LIN {X 0,Y 293.963,Z 864.101,A -85,B 0,C 180,E1 22484.69,E2 22484.69} C_VEL
LIN {X 0,Y 291.731,Z 885.512,A -85,B 0,C 180,E1 22491.042,E2 22491.042} C_VEL
LIN {X 0,Y 291.359,Z 899.593,A -85,B 0,C 180,E1 22497.023,E2 22497.023} C_VEL
LIN {X 0,Y 292.208,Z 908.654,A -85,B 0,C 180,E1 22502.975,E2 22502.975} C_VEL
LIN {X 0,Y 295.422,Z 913.131,A -85,B 0,C 180,E1 22508.853,E2 22508.853} C_VEL
LIN {X 0,Y 300.698,Z 913.398,A -85,B 0,C 180,E1 22514.593,E2 22514.593} C_VEL
LIN {X 0,Y 310.967,Z 908.328,A -85,B 0,C 180,E1 22521.434,E2 22521.434} C_VEL
LIN {X 0,Y 325.668,Z 897.626,A -85,B 0,C 180,E1 22527.724,E2 22527.724} C_VEL
LIN {X 0,Y 349.66,Z 878.572,A -85,B 0,C 180,E1 22534.282,E2 22534.282} C_VEL
LIN {X 0,Y 365.291,Z 866.098,A -85,B 0,C 180,E1 22537.259,E2 22537.259} C_VEL
LIN {X 0,Y 331.443,Z 903.67,A -85,B 0,C 180,E1 22545.054,E2 22545.054} C_VEL
LIN {X 0,Y 310.197,Z 930.316,A -85,B 0,C 180,E1 22553.256,E2 22553.256} C_VEL
LIN {X 0,Y 296.493,Z 951.276,A -85,B 0,C 180,E1 22562.626,E2 22562.626} C_VEL
LIN {X 0,Y 290.643,Z 964.921,A -85,B 0,C 180,E1 22571.781,E2 22571.781} C_VEL
LIN {X 0,Y 289.464,Z 970.796,A -85,B 0,C 180,E1 22577.922,E2 22577.922} C_VEL
LIN {X 0,Y 289.713,Z 973.891,A -85,B 0,C 180,E1 22584.004,E2 22584.004} C_VEL
LIN {X 0,Y 290.557,Z 973.915,A -85,B 0,C 180,E1 22590.008,E2 22590.008} C_VEL
LIN {X 0,Y 290.157,Z 969.252,A -85,B 0,C 180,E1 22597.235,E2 22597.235} C_VEL
LIN {X 0,Y 290.402,Z 960.92,A -85,B 0,C 180,E1 22605.131,E2 22605.131} C_VEL
LIN {X 0,Y 292.996,Z 947.16,A -85,B 0,C 180,E1 22612.83,E2 22612.83} C_VEL
LIN {X 0,Y 298.847,Z 927.81,A -85,B 0,C 180,E1 22620.054,E2 22620.054} C_VEL
LIN {X 0,Y 307.221,Z 903.866,A -85,B 0,C 180,E1 22626.297,E2 22626.297} C_VEL
LIN {X 0,Y 316.929,Z 875.444,A -85,B 0,C 180,E1 22631.566,E2 22631.566} C_VEL
LIN {X 0,Y 326.727,Z 843.194,A -85,B 0,C 180,E1 22635.791,E2 22635.791} C_VEL
LIN {X 0,Y 335.469,Z 807.511,A -85,B 0,C 180,E1 22639.019,E2 22639.019} C_VEL
LIN {X 0,Y 345.478,Z 755.854,A -85,B 0,C 180,E1 22642.286,E2 22642.286} C_VEL
LIN {X 0,Y 347.447,Z 742.622,A -85,B 0,C 180,E1 22643.014,E2 22643.014} C_VEL
LIN {X 0,Y 330.365,Z 668.326,A -85,B 0,C 180,E1 22652.795,E2 22652.795} C_VEL
LIN {X 0,Y 328.166,Z 660.053,A -85,B 0,C 180,E1 22654.078,E2 22654.078} C_VEL
LIN {X 0,Y 318.814,Z 645.104,A -85,B 0,C 180,E1 22658.71,E2 22658.71} C_VEL
LIN {X 0,Y 315.788,Z 643.613,A -85,B 0,C 180,E1 22660.163,E2 22660.163} C_VEL
LIN {X 0,Y 310.485,Z 643.76,A -85,B 0,C 180,E1 22662.744,E2 22662.744} C_VEL
LIN {X 0,Y 306.565,Z 637.974,A -85,B 0,C 180,E1 22665.692,E2 22665.692} C_VEL
LIN {X 0,Y 302.237,Z 631.324,A -85,B 0,C 180,E1 22669.893,E2 22669.893} C_VEL
LIN {X 0,Y 298.732,Z 625.168,A -85,B 0,C 180,E1 22675.361,E2 22675.361} C_VEL
LIN {X 0,Y 297.1,Z 623.883,A -85,B 0,C 180,E1 22683.651,E2 22683.651} C_VEL
LIN {X 0,Y 298.132,Z 625.461,A -85,B 0,C 180,E1 22687.753,E2 22687.753} C_VEL
LIN {X 0,Y 301.609,Z 631.309,A -85,B 0,C 180,E1 22693.761,E2 22693.761} C_VEL
LIN {X 0,Y 306.971,Z 640.946,A -85,B 0,C 180,E1 22699.364,E2 22699.364} C_VEL
LIN {X 0,Y 313.809,Z 652.315,A -85,B 0,C 180,E1 22704.391,E2 22704.391} C_VEL
LIN {X 0,Y 324.604,Z 672.136,A -85,B 0,C 180,E1 22710.592,E2 22710.592} C_VEL
LIN {X 0,Y 335.868,Z 696.454,A -85,B 0,C 180,E1 22715.988,E2 22715.988} C_VEL
LIN {X 0,Y 344.416,Z 721.512,A -85,B 0,C 180,E1 22720.282,E2 22720.282} C_VEL
LIN {X 0,Y 347.289,Z 737.002,A -85,B 0,C 180,E1 22722.591,E2 22722.591} C_VEL
LIN {X 0,Y 337.653,Z 771.94,A -85,B 0,C 180,E1 22725.601,E2 22725.601} C_VEL
LIN {X 0,Y 326.46,Z 803.597,A -85,B 0,C 180,E1 22729.465,E2 22729.465} C_VEL
LIN {X 0,Y 314.714,Z 831.598,A -85,B 0,C 180,E1 22734.275,E2 22734.275} C_VEL
LIN {X 0,Y 303.549,Z 855.386,A -85,B 0,C 180,E1 22740.046,E2 22740.046} C_VEL
LIN {X 0,Y 294.509,Z 873.806,A -85,B 0,C 180,E1 22746.493,E2 22746.493} C_VEL
LIN {X 0,Y 287.852,Z 887.888,A -85,B 0,C 180,E1 22753.949,E2 22753.949} C_VEL
LIN {X 0,Y 284.529,Z 895.556,A -85,B 0,C 180,E1 22760.799,E2 22760.799} C_VEL
LIN {X 0,Y 283.36,Z 898.747,A -85,B 0,C 180,E1 22766.926,E2 22766.926} C_VEL
LIN {X 0,Y 283.471,Z 898.702,A -85,B 0,C 180,E1 22773.056,E2 22773.056} C_VEL
LIN {X 0,Y 285.219,Z 893.795,A -85,B 0,C 180,E1 22781.036,E2 22781.036} C_VEL
LIN {X 0,Y 290.075,Z 882.965,A -85,B 0,C 180,E1 22788.94,E2 22788.94} C_VEL
LIN {X 0,Y 297.256,Z 868.058,A -85,B 0,C 180,E1 22795.666,E2 22795.666} C_VEL
LIN {X 0,Y 307.265,Z 847.474,A -85,B 0,C 180,E1 22802.004,E2 22802.004} C_VEL
LIN {X 0,Y 319.289,Z 820.866,A -85,B 0,C 180,E1 22807.652,E2 22807.652} C_VEL
LIN {X 0,Y 331.221,Z 790.376,A -85,B 0,C 180,E1 22812.204,E2 22812.204} C_VEL
LIN {X 0,Y 342.367,Z 755.645,A -85,B 0,C 180,E1 22815.832,E2 22815.832} C_VEL
LIN {X 0,Y 347.152,Z 734.437,A -85,B 0,C 180,E1 22817.597,E2 22817.597} C_VEL
LIN {X 0,Y 340.844,Z 709.744,A -85,B 0,C 180,E1 22821.525,E2 22821.525} C_VEL
LIN {X 0,Y 338.651,Z 705.006,A -85,B 0,C 180,E1 22822.452,E2 22822.452} C_VEL
LIN {X 0,Y 327.156,Z 719.096,A -85,B 0,C 180,E1 22823.933,E2 22823.933} C_VEL
LIN {X 0,Y 319.775,Z 728.865,A -85,B 0,C 180,E1 22824.78,E2 22824.78} C_VEL
LIN {X 0,Y 316.357,Z 731.37,A -85,B 0,C 180,E1 22825.427,E2 22825.427} C_VEL
LIN {X 0,Y 310.131,Z 739.58,A -85,B 0,C 180,E1 22826.143,E2 22826.143} C_VEL
LIN {X 0,Y 305.98,Z 742.075,A -85,B 0,C 180,E1 22827.121,E2 22827.121} C_VEL
LIN {X 0,Y 299.689,Z 781.3,A -85,B 0,C 180,E1 22830.684,E2 22830.684} C_VEL
LIN {X 0,Y 293.509,Z 817.551,A -85,B 0,C 180,E1 22835.353,E2 22835.353} C_VEL
LIN {X 0,Y 288.411,Z 848.674,A -85,B 0,C 180,E1 22840.89,E2 22840.89} C_VEL
LIN {X 0,Y 284.991,Z 873.356,A -85,B 0,C 180,E1 22846.948,E2 22846.948} C_VEL
LIN {X 0,Y 283.545,Z 891.452,A -85,B 0,C 180,E1 22853.1,E2 22853.1} C_VEL
LIN {X 0,Y 283.712,Z 905.176,A -85,B 0,C 180,E1 22860.004,E2 22860.004} C_VEL
LIN {X 0,Y 285.808,Z 912.321,A -85,B 0,C 180,E1 22866.089,E2 22866.089} C_VEL
LIN {X 0,Y 290.137,Z 915.158,A -85,B 0,C 180,E1 22872.059,E2 22872.059} C_VEL
LIN {X 0,Y 296.986,Z 913.91,A -85,B 0,C 180,E1 22877.825,E2 22877.825} C_VEL
LIN {X 0,Y 309.514,Z 907.303,A -85,B 0,C 180,E1 22884.588,E2 22884.588} C_VEL
LIN {X 0,Y 328.712,Z 894.071,A -85,B 0,C 180,E1 22891.233,E2 22891.233} C_VEL
LIN {X 0,Y 355.231,Z 874.877,A -85,B 0,C 180,E1 22897.074,E2 22897.074} C_VEL
LIN {X 0,Y 355.139,Z 875.264,A -85,B 0,C 180,E1 22897.5,E2 22897.5} C_VEL
LIN {X 0,Y 325.035,Z 906.212,A -85,B 0,C 180,E1 22904.36,E2 22904.36} C_VEL
LIN {X 0,Y 302.368,Z 932.529,A -85,B 0,C 180,E1 22913.044,E2 22913.044} C_VEL
LIN {X 0,Y 288.301,Z 952.616,A -85,B 0,C 180,E1 22922.819,E2 22922.819} C_VEL
LIN {X 0,Y 282.424,Z 965.885,A -85,B 0,C 180,E1 22932.847,E2 22932.847} C_VEL
LIN {X 0,Y 281.639,Z 971.637,A -85,B 0,C 180,E1 22940.721,E2 22940.721} C_VEL
LIN {X 0,Y 282.269,Z 973.069,A -85,B 0,C 180,E1 22946.931,E2 22946.931} C_VEL
LIN {X 0,Y 282.753,Z 972.61,A -85,B 0,C 180,E1 22950.008,E2 22950.008} C_VEL
LIN {X 0,Y 282.308,Z 968.072,A -85,B 0,C 180,E1 22957.437,E2 22957.437} C_VEL
LIN {X 0,Y 282.57,Z 959.86,A -85,B 0,C 180,E1 22965.561,E2 22965.561} C_VEL
LIN {X 0,Y 285.43,Z 946.05,A -85,B 0,C 180,E1 22973.471,E2 22973.471} C_VEL
LIN {X 0,Y 291.695,Z 926.652,A -85,B 0,C 180,E1 22980.87,E2 22980.87} C_VEL
LIN {X 0,Y 300.52,Z 902.658,A -85,B 0,C 180,E1 22987.241,E2 22987.241} C_VEL
LIN {X 0,Y 310.747,Z 874.204,A -85,B 0,C 180,E1 22992.585,E2 22992.585} C_VEL
LIN {X 0,Y 320.997,Z 841.931,A -85,B 0,C 180,E1 22996.853,E2 22996.853} C_VEL
LIN {X 0,Y 330.033,Z 806.731,A -85,B 0,C 180,E1 23000.051,E2 23000.051} C_VEL
LIN {X 0,Y 340.278,Z 755.895,A -85,B 0,C 180,E1 23003.286,E2 23003.286} C_VEL
LIN {X 0,Y 341.629,Z 744.601,A -85,B 0,C 180,E1 23003.994,E2 23003.994} C_VEL
LIN {X 0,Y 326.511,Z 673.546,A -85,B 0,C 180,E1 23013.593,E2 23013.593} C_VEL
LIN {X 0,Y 324.558,Z 665.67,A -85,B 0,C 180,E1 23014.887,E2 23014.887} C_VEL
LIN {X 0,Y 314.172,Z 649.402,A -85,B 0,C 180,E1 23020.362,E2 23020.362} C_VEL
LIN {X 0,Y 310.485,Z 643.76,A -85,B 0,C 180,E1 23022.744,E2 23022.744} C_VEL
LIN {X 0,Y 305.445,Z 642.335,A -85,B 0,C 180,E1 23025.87,E2 23025.87} C_VEL
LIN {X 0,Y 301.668,Z 640.672,A -85,B 0,C 180,E1 23028.861,E2 23028.861} C_VEL
LIN {X 0,Y 301.51,Z 640.292,A -85,B 0,C 180,E1 23029.053,E2 23029.053} C_VEL
LIN {X 0,Y 297.03,Z 632.389,A -85,B 0,C 180,E1 23035.884,E2 23035.884} C_VEL
LIN {X 0,Y 296.025,Z 631.913,A -85,B 0,C 180,E1 23045.871,E2 23045.871} C_VEL
LIN {X 0,Y 296.469,Z 633.916,A -85,B 0,C 180,E1 23047.982,E2 23047.982} C_VEL
LIN {X 0,Y 300.315,Z 640.431,A -85,B 0,C 180,E1 23054.409,E2 23054.409} C_VEL
LIN {X 0,Y 304.755,Z 648.592,A -85,B 0,C 180,E1 23059.15,E2 23059.15} C_VEL
LIN {X 0,Y 311.109,Z 659.692,A -85,B 0,C 180,E1 23064.063,E2 23064.063} C_VEL
LIN {X 0,Y 321.105,Z 678.543,A -85,B 0,C 180,E1 23070.055,E2 23070.055} C_VEL
LIN {X 0,Y 331.913,Z 702.757,A -85,B 0,C 180,E1 23075.512,E2 23075.512} C_VEL
LIN {X 0,Y 339.614,Z 727.51,A -85,B 0,C 180,E1 23079.862,E2 23079.862} C_VEL
LIN {X 0,Y 341.411,Z 740.531,A -85,B 0,C 180,E1 23081.817,E2 23081.817} C_VEL
LIN {X 0,Y 331.408,Z 775.162,A -85,B 0,C 180,E1 23084.883,E2 23084.883} C_VEL
LIN {X 0,Y 319.916,Z 806.201,A -85,B 0,C 180,E1 23088.789,E2 23088.789} C_VEL
LIN {X 0,Y 307.632,Z 834.289,A -85,B 0,C 180,E1 23093.759,E2 23093.759} C_VEL
LIN {X 0,Y 295.696,Z 858.447,A -85,B 0,C 180,E1 23099.906,E2 23099.906} C_VEL
LIN {X 0,Y 286.434,Z 876.562,A -85,B 0,C 180,E1 23106.616,E2 23106.616} C_VEL
LIN {X 0,Y 279.777,Z 889.923,A -85,B 0,C 180,E1 23114.28,E2 23114.28} C_VEL
LIN {X 0,Y 276.772,Z 896.554,A -85,B 0,C 180,E1 23120.538,E2 23120.538} C_VEL
LIN {X 0,Y 275.54,Z 899.735,A -85,B 0,C 180,E1 23126.839,E2 23126.839} C_VEL
LIN {X 0,Y 275.65,Z 899.69,A -85,B 0,C 180,E1 23133.142,E2 23133.142} C_VEL
LIN {X 0,Y 277.381,Z 895.05,A -85,B 0,C 180,E1 23141.06,E2 23141.06} C_VEL
LIN {X 0,Y 282.091,Z 885.159,A -85,B 0,C 180,E1 23148.792,E2 23148.792} C_VEL
LIN {X 0,Y 290.171,Z 869.098,A -85,B 0,C 180,E1 23156.341,E2 23156.341} C_VEL
LIN {X 0,Y 301.279,Z 847.128,A -85,B 0,C 180,E1 23163.147,E2 23163.147} C_VEL
LIN {X 0,Y 313.878,Z 820.133,A -85,B 0,C 180,E1 23168.86,E2 23168.86} C_VEL
LIN {X 0,Y 326.366,Z 788.955,A -85,B 0,C 180,E1 23173.438,E2 23173.438} C_VEL
LIN {X 0,Y 337.493,Z 754.65,A -85,B 0,C 180,E1 23176.963,E2 23176.963} C_VEL
LIN {X 0,Y 341.605,Z 738.117,A -85,B 0,C 180,E1 23178.307,E2 23178.307} C_VEL
LIN {X 0,Y 336.717,Z 716.824,A -85,B 0,C 180,E1 23181.789,E2 23181.789} C_VEL
LIN {X 0,Y 335.916,Z 715.7,A -85,B 0,C 180,E1 23182.092,E2 23182.092} C_VEL
LIN {X 0,Y 329.302,Z 723.742,A -85,B 0,C 180,E1 23182.863,E2 23182.863} C_VEL
LIN {X 0,Y 320.621,Z 734.521,A -85,B 0,C 180,E1 23183.806,E2 23183.806} C_VEL
LIN {X 0,Y 314.182,Z 741.259,A -85,B 0,C 180,E1 23184.652,E2 23184.652} C_VEL
LIN {X 0,Y 307.063,Z 747.905,A -85,B 0,C 180,E1 23185.758,E2 23185.758} C_VEL
LIN {X 0,Y 299.477,Z 755.381,A -85,B 0,C 180,E1 23186.895,E2 23186.895} C_VEL
LIN {X 0,Y 296.238,Z 757.549,A -85,B 0,C 180,E1 23187.839,E2 23187.839} C_VEL
LIN {X 0,Y 289.52,Z 796.999,A -85,B 0,C 180,E1 23192.06,E2 23192.06} C_VEL
LIN {X 0,Y 283.552,Z 831.369,A -85,B 0,C 180,E1 23197.216,E2 23197.216} C_VEL
LIN {X 0,Y 278.964,Z 859.516,A -85,B 0,C 180,E1 23203.033,E2 23203.033} C_VEL
LIN {X 0,Y 276.333,Z 881.753,A -85,B 0,C 180,E1 23209.342,E2 23209.342} C_VEL
LIN {X 0,Y 275.548,Z 898.545,A -85,B 0,C 180,E1 23216.063,E2 23216.063} C_VEL
LIN {X 0,Y 276.484,Z 909.926,A -85,B 0,C 180,E1 23223.145,E2 23223.145} C_VEL
LIN {X 0,Y 279.977,Z 915.293,A -85,B 0,C 180,E1 23229.346,E2 23229.346} C_VEL
LIN {X 0,Y 285.775,Z 916.584,A -85,B 0,C 180,E1 23235.374,E2 23235.374} C_VEL
LIN {X 0,Y 296.93,Z 912.826,A -85,B 0,C 180,E1 23242.501,E2 23242.501} C_VEL
LIN {X 0,Y 314.72,Z 902.755,A -85,B 0,C 180,E1 23249.567,E2 23249.567} C_VEL
LIN {X 0,Y 340.531,Z 885.96,A -85,B 0,C 180,E1 23256.034,E2 23256.034} C_VEL
LIN {X 0,Y 346.696,Z 881.931,A -85,B 0,C 180,E1 23257.183,E2 23257.183} C_VEL
LIN {X 0,Y 312.804,Z 914.491,A -85,B 0,C 180,E1 23265.393,E2 23265.393} C_VEL
LIN {X 0,Y 290.43,Z 939.321,A -85,B 0,C 180,E1 23274.989,E2 23274.989} C_VEL
LIN {X 0,Y 278.434,Z 956.654,A -85,B 0,C 180,E1 23285.065,E2 23285.065} C_VEL
LIN {X 0,Y 274.025,Z 967.466,A -85,B 0,C 180,E1 23295.168,E2 23295.168} C_VEL
LIN {X 0,Y 274.019,Z 971.558,A -85,B 0,C 180,E1 23303.659,E2 23303.659} C_VEL
LIN {X 0,Y 274.983,Z 971.26,A -85,B 0,C 180,E1 23310.009,E2 23310.009} C_VEL
LIN {X 0,Y 274.418,Z 966.967,A -85,B 0,C 180,E1 23317.783,E2 23317.783} C_VEL
LIN {X 0,Y 274.735,Z 958.801,A -85,B 0,C 180,E1 23326.016,E2 23326.016} C_VEL
LIN {X 0,Y 277.873,Z 944.933,A -85,B 0,C 180,E1 23334.149,E2 23334.149} C_VEL
LIN {X 0,Y 284.342,Z 926.124,A -85,B 0,C 180,E1 23341.516,E2 23341.516} C_VEL
LIN {X 0,Y 293.926,Z 901.439,A -85,B 0,C 180,E1 23348.225,E2 23348.225} C_VEL
LIN {X 0,Y 304.675,Z 872.948,A -85,B 0,C 180,E1 23353.643,E2 23353.643} C_VEL
LIN {X 0,Y 315.422,Z 840.584,A -85,B 0,C 180,E1 23357.956,E2 23357.956} C_VEL
LIN {X 0,Y 324.619,Z 806.394,A -85,B 0,C 180,E1 23361.084,E2 23361.084} C_VEL
LIN {X 0,Y 335.497,Z 754.329,A -85,B 0,C 180,E1 23364.396,E2 23364.396} C_VEL
LIN {X 0,Y 336.175,Z 747.644,A -85,B 0,C 180,E1 23364.852,E2 23364.852} C_VEL
LIN {X 0,Y 322.845,Z 679.483,A -85,B 0,C 180,E1 23374.297,E2 23374.297} C_VEL
LIN {X 0,Y 320.939,Z 671.429,A -85,B 0,C 180,E1 23375.641,E2 23375.641} C_VEL
LIN {X 0,Y 309.444,Z 652.358,A -85,B 0,C 180,E1 23382.382,E2 23382.382} C_VEL
LIN {X 0,Y 303.923,Z 644.729,A -85,B 0,C 180,E1 23386.576,E2 23386.576} C_VEL
LIN {X 0,Y 301.51,Z 640.292,A -85,B 0,C 180,E1 23389.053,E2 23389.053} C_VEL
LIN {X 0,Y 299.597,Z 640.524,A -85,B 0,C 180,E1 23390.668,E2 23390.668} C_VEL
LIN {X 0,Y 296.515,Z 643.952,A -85,B 0,C 180,E1 23393.147,E2 23393.147} C_VEL
LIN {X 0,Y 296.313,Z 643.797,A -85,B 0,C 180,E1 23393.435,E2 23393.435} C_VEL
LIN {X 0,Y 294.879,Z 639.708,A -85,B 0,C 180,E1 23397.052,E2 23397.052} C_VEL
LIN {X 0,Y 294.554,Z 640.25,A -85,B 0,C 180,E1 23406.919,E2 23406.919} C_VEL
LIN {X 0,Y 298.182,Z 648.151,A -85,B 0,C 180,E1 23414.218,E2 23414.218} C_VEL
LIN {X 0,Y 302.552,Z 656.224,A -85,B 0,C 180,E1 23418.965,E2 23418.965} C_VEL
LIN {X 0,Y 310.3,Z 670.155,A -85,B 0,C 180,E1 23424.995,E2 23424.995} C_VEL
LIN {X 0,Y 320.367,Z 691.113,A -85,B 0,C 180,E1 23431.099,E2 23431.099} C_VEL
LIN {X 0,Y 329.994,Z 715.209,A -85,B 0,C 180,E1 23436.227,E2 23436.227} C_VEL
LIN {X 0,Y 335.936,Z 740.581,A -85,B 0,C 180,E1 23440.621,E2 23440.621} C_VEL
LIN {X 0,Y 332.723,Z 754.359,A -85,B 0,C 180,E1 23441.83,E2 23441.83} C_VEL
LIN {X 0,Y 321.104,Z 789.415,A -85,B 0,C 180,E1 23445.409,E2 23445.409} C_VEL
LIN {X 0,Y 308.323,Z 820.439,A -85,B 0,C 180,E1 23449.981,E2 23449.981} C_VEL
LIN {X 0,Y 295.394,Z 847.143,A -85,B 0,C 180,E1 23455.641,E2 23455.641} C_VEL
LIN {X 0,Y 284.158,Z 868.467,A -85,B 0,C 180,E1 23462.178,E2 23462.178} C_VEL
LIN {X 0,Y 275.343,Z 884.758,A -85,B 0,C 180,E1 23469.727,E2 23469.727} C_VEL
LIN {X 0,Y 270.333,Z 894.669,A -85,B 0,C 180,E1 23477.035,E2 23477.035} C_VEL
LIN {X 0,Y 268.15,Z 899.522,A -85,B 0,C 180,E1 23483.502,E2 23483.502} C_VEL
LIN {X 0,Y 267.775,Z 901.131,A -85,B 0,C 180,E1 23489.991,E2 23489.991} C_VEL
LIN {X 0,Y 268.224,Z 899.464,A -85,B 0,C 180,E1 23496.478,E2 23496.478} C_VEL
LIN {X 0,Y 271.288,Z 892.82,A -85,B 0,C 180,E1 23504.547,E2 23504.547} C_VEL
LIN {X 0,Y 277.595,Z 880.506,A -85,B 0,C 180,E1 23512.453,E2 23512.453} C_VEL
LIN {X 0,Y 287.56,Z 861.943,A -85,B 0,C 180,E1 23519.977,E2 23519.977} C_VEL
LIN {X 0,Y 299.842,Z 838.082,A -85,B 0,C 180,E1 23526.397,E2 23526.397} C_VEL
LIN {X 0,Y 312.256,Z 811.181,A -85,B 0,C 180,E1 23531.438,E2 23531.438} C_VEL
LIN {X 0,Y 324.825,Z 778.911,A -85,B 0,C 180,E1 23535.688,E2 23535.688} C_VEL
LIN {X 0,Y 335.426,Z 743.926,A -85,B 0,C 180,E1 23538.895,E2 23538.895} C_VEL
LIN {X 0,Y 335.302,Z 736.78,A -85,B 0,C 180,E1 23539.849,E2 23539.849} C_VEL
LIN {X 0,Y 332.931,Z 726.038,A -85,B 0,C 180,E1 23541.693,E2 23541.693} C_VEL
LIN {X 0,Y 322.621,Z 738.908,A -85,B 0,C 180,E1 23542.667,E2 23542.667} C_VEL
LIN {X 0,Y 307.588,Z 753.393,A -85,B 0,C 180,E1 23544.646,E2 23544.646} C_VEL
LIN {X 0,Y 298.305,Z 761.782,A -85,B 0,C 180,E1 23546.044,E2 23546.044} C_VEL
LIN {X 0,Y 294.774,Z 764.171,A -85,B 0,C 180,E1 23546.75,E2 23546.75} C_VEL
LIN {X 0,Y 289.618,Z 768.793,A -85,B 0,C 180,E1 23547.569,E2 23547.569} C_VEL
LIN {X 0,Y 286.619,Z 770.796,A -85,B 0,C 180,E1 23548.543,E2 23548.543} C_VEL
LIN {X 0,Y 279.985,Z 808.372,A -85,B 0,C 180,E1 23553.116,E2 23553.116} C_VEL
LIN {X 0,Y 274.281,Z 840.385,A -85,B 0,C 180,E1 23558.541,E2 23558.541} C_VEL
LIN {X 0,Y 270.036,Z 868.042,A -85,B 0,C 180,E1 23564.966,E2 23564.966} C_VEL
LIN {X 0,Y 267.905,Z 889.543,A -85,B 0,C 180,E1 23571.973,E2 23571.973} C_VEL
LIN {X 0,Y 267.866,Z 904.645,A -85,B 0,C 180,E1 23579.194,E2 23579.194} C_VEL
LIN {X 0,Y 270.192,Z 913.939,A -85,B 0,C 180,E1 23586.442,E2 23586.442} C_VEL
LIN {X 0,Y 274.927,Z 917.659,A -85,B 0,C 180,E1 23592.737,E2 23592.737} C_VEL
LIN {X 0,Y 282.404,Z 917.539,A -85,B 0,C 180,E1 23598.779,E2 23598.779} C_VEL
LIN {X 0,Y 295.992,Z 912.372,A -85,B 0,C 180,E1 23605.791,E2 23605.791} C_VEL
LIN {X 0,Y 316.583,Z 901.259,A -85,B 0,C 180,E1 23612.574,E2 23612.574} C_VEL
LIN {X 0,Y 335.318,Z 890.227,A -85,B 0,C 180,E1 23616.783,E2 23616.783} C_VEL
LIN {X 0,Y 336.215,Z 889.95,A -85,B 0,C 180,E1 23617.359,E2 23617.359} C_VEL
LIN {X 0,Y 303.371,Z 919.431,A -85,B 0,C 180,E1 23625.645,E2 23625.645} C_VEL
LIN {X 0,Y 280.056,Z 943.79,A -85,B 0,C 180,E1 23636.33,E2 23636.33} C_VEL
LIN {X 0,Y 269.246,Z 959.185,A -85,B 0,C 180,E1 23646.81,E2 23646.81} C_VEL
LIN {X 0,Y 265.962,Z 967.867,A -85,B 0,C 180,E1 23656.837,E2 23656.837} C_VEL
LIN {X 0,Y 266.156,Z 970.372,A -85,B 0,C 180,E1 23663.471,E2 23663.471} C_VEL
LIN {X 0,Y 267.189,Z 969.885,A -85,B 0,C 180,E1 23670.009,E2 23670.009} C_VEL
LIN {X 0,Y 266.513,Z 965.846,A -85,B 0,C 180,E1 23678.18,E2 23678.18} C_VEL
LIN {X 0,Y 266.947,Z 957.741,A -85,B 0,C 180,E1 23686.497,E2 23686.497} C_VEL
LIN {X 0,Y 270.351,Z 943.817,A -85,B 0,C 180,E1 23694.866,E2 23694.866} C_VEL
LIN {X 0,Y 277.545,Z 924.309,A -85,B 0,C 180,E1 23702.635,E2 23702.635} C_VEL
LIN {X 0,Y 287.87,Z 899.247,A -85,B 0,C 180,E1 23709.474,E2 23709.474} C_VEL
LIN {X 0,Y 299.144,Z 870.519,A -85,B 0,C 180,E1 23714.934,E2 23714.934} C_VEL
LIN {X 0,Y 310.48,Z 837.558,A -85,B 0,C 180,E1 23719.28,E2 23719.28} C_VEL
LIN {X 0,Y 320.285,Z 801.776,A -85,B 0,C 180,E1 23722.479,E2 23722.479} C_VEL
LIN {X 0,Y 330.764,Z 750.703,A -85,B 0,C 180,E1 23725.746,E2 23725.746} C_VEL
LIN {X 0,Y 318.395,Z 680.031,A -85,B 0,C 180,E1 23735.792,E2 23735.792} C_VEL
LIN {X 0,Y 311.902,Z 668.09,A -85,B 0,C 180,E1 23739.495,E2 23739.495} C_VEL
LIN {X 0,Y 304.847,Z 656.769,A -85,B 0,C 180,E1 23744.32,E2 23744.32} C_VEL
LIN {X 0,Y 298.811,Z 646.648,A -85,B 0,C 180,E1 23750.164,E2 23750.164} C_VEL
LIN {X 0,Y 296.313,Z 643.797,A -85,B 0,C 180,E1 23753.435,E2 23753.435} C_VEL
LIN {X 0,Y 294.006,Z 644.534,A -85,B 0,C 180,E1 23756.816,E2 23756.816} C_VEL
LIN {X 0,Y 292.311,Z 646.881,A -85,B 0,C 180,E1 23760.263,E2 23760.263} C_VEL
LIN {X 0,Y 292.729,Z 648.25,A -85,B 0,C 180,E1 23766.869,E2 23766.869} C_VEL
LIN {X 0,Y 296.03,Z 655.643,A -85,B 0,C 180,E1 23773.902,E2 23773.902} C_VEL
LIN {X 0,Y 300.398,Z 664.131,A -85,B 0,C 180,E1 23778.94,E2 23778.94} C_VEL
LIN {X 0,Y 307.709,Z 678.202,A -85,B 0,C 180,E1 23784.882,E2 23784.882} C_VEL
LIN {X 0,Y 316.725,Z 697.539,A -85,B 0,C 180,E1 23790.582,E2 23790.582} C_VEL
LIN {X 0,Y 325.377,Z 720.425,A -85,B 0,C 180,E1 23795.585,E2 23795.585} C_VEL
LIN {X 0,Y 330.488,Z 744.596,A -85,B 0,C 180,E1 23799.917,E2 23799.917} C_VEL
LIN {X 0,Y 319.393,Z 780.406,A -85,B 0,C 180,E1 23803.233,E2 23803.233} C_VEL
LIN {X 0,Y 306.72,Z 811.783,A -85,B 0,C 180,E1 23807.399,E2 23807.399} C_VEL
LIN {X 0,Y 293.215,Z 839.992,A -85,B 0,C 180,E1 23812.766,E2 23812.766} C_VEL
LIN {X 0,Y 280.777,Z 863.157,A -85,B 0,C 180,E1 23819.15,E2 23819.15} C_VEL
LIN {X 0,Y 270.247,Z 881.725,A -85,B 0,C 180,E1 23826.882,E2 23826.882} C_VEL
LIN {X 0,Y 263.628,Z 893.953,A -85,B 0,C 180,E1 23835.001,E2 23835.001} C_VEL
LIN {X 0,Y 260.355,Z 900.513,A -85,B 0,C 180,E1 23843.307,E2 23843.307} C_VEL
LIN {X 0,Y 259.951,Z 902.117,A -85,B 0,C 180,E1 23849.991,E2 23849.991} C_VEL
LIN {X 0,Y 260.426,Z 900.459,A -85,B 0,C 180,E1 23856.673,E2 23856.673} C_VEL
LIN {X 0,Y 263.691,Z 893.824,A -85,B 0,C 180,E1 23864.976,E2 23864.976} C_VEL
LIN {X 0,Y 270.324,Z 881.522,A -85,B 0,C 180,E1 23873.092,E2 23873.092} C_VEL
LIN {X 0,Y 280.843,Z 862.846,A -85,B 0,C 180,E1 23880.822,E2 23880.822} C_VEL
LIN {X 0,Y 293.491,Z 839.273,A -85,B 0,C 180,E1 23887.278,E2 23887.278} C_VEL
LIN {X 0,Y 306.953,Z 811,A -85,B 0,C 180,E1 23892.604,E2 23892.604} C_VEL
LIN {X 0,Y 319.933,Z 778.501,A -85,B 0,C 180,E1 23896.851,E2 23896.851} C_VEL
LIN {X 0,Y 330.373,Z 743.786,A -85,B 0,C 180,E1 23900.067,E2 23900.067} C_VEL
LIN {X 0,Y 329.475,Z 738.256,A -85,B 0,C 180,E1 23901.025,E2 23901.025} C_VEL
LIN {X 0,Y 308.569,Z 758.46,A -85,B 0,C 180,E1 23903.473,E2 23903.473} C_VEL
LIN {X 0,Y 296.826,Z 768.185,A -85,B 0,C 180,E1 23905.2,E2 23905.2} C_VEL
LIN {X 0,Y 289.169,Z 774.312,A -85,B 0,C 180,E1 23906.453,E2 23906.453} C_VEL
LIN {X 0,Y 283.133,Z 778.426,A -85,B 0,C 180,E1 23907.658,E2 23907.658} C_VEL
LIN {X 0,Y 278.044,Z 781.639,A -85,B 0,C 180,E1 23908.834,E2 23908.834} C_VEL
LIN {X 0,Y 277.277,Z 781.954,A -85,B 0,C 180,E1 23909.194,E2 23909.194} C_VEL
LIN {X 0,Y 270.464,Z 818.842,A -85,B 0,C 180,E1 23914.278,E2 23914.278} C_VEL
LIN {X 0,Y 264.945,Z 849.911,A -85,B 0,C 180,E1 23920.199,E2 23920.199} C_VEL
LIN {X 0,Y 261.235,Z 875.777,A -85,B 0,C 180,E1 23927.019,E2 23927.019} C_VEL
LIN {X 0,Y 259.808,Z 895.102,A -85,B 0,C 180,E1 23934.148,E2 23934.148} C_VEL
LIN {X 0,Y 260.326,Z 908.802,A -85,B 0,C 180,E1 23941.672,E2 23941.672} C_VEL
LIN {X 0,Y 264.567,Z 917.29,A -85,B 0,C 180,E1 23949.895,E2 23949.895} C_VEL
LIN {X 0,Y 270.844,Z 919.496,A -85,B 0,C 180,E1 23956.244,E2 23956.244} C_VEL
LIN {X 0,Y 282.978,Z 917.21,A -85,B 0,C 180,E1 23963.676,E2 23963.676} C_VEL
LIN {X 0,Y 300.096,Z 909.984,A -85,B 0,C 180,E1 23970.322,E2 23970.322} C_VEL
LIN {X 0,Y 327.208,Z 895.903,A -85,B 0,C 180,E1 23977.008,E2 23977.008} C_VEL
LIN {X 0,Y 291.64,Z 925.855,A -85,B 0,C 180,E1 23986.658,E2 23986.658} C_VEL
LIN {X 0,Y 270.848,Z 946.526,A -85,B 0,C 180,E1 23997.039,E2 23997.039} C_VEL
LIN {X 0,Y 260.238,Z 961.124,A -85,B 0,C 180,E1 24008.663,E2 24008.663} C_VEL
LIN {X 0,Y 258.12,Z 966.893,A -85,B 0,C 180,E1 24016.429,E2 24016.429} C_VEL
LIN {X 0,Y 258.48,Z 969.285,A -85,B 0,C 180,E1 24025.135,E2 24025.135} C_VEL
LIN {X 0,Y 259.416,Z 968.496,A -85,B 0,C 180,E1 24030.009,E2 24030.009} C_VEL
LIN {X 0,Y 258.642,Z 964.833,A -85,B 0,C 180,E1 24038.431,E2 24038.431} C_VEL
LIN {X 0,Y 259.159,Z 956.68,A -85,B 0,C 180,E1 24047.007,E2 24047.007} C_VEL
LIN {X 0,Y 262.895,Z 942.712,A -85,B 0,C 180,E1 24055.621,E2 24055.621} C_VEL
LIN {X 0,Y 270.57,Z 923.24,A -85,B 0,C 180,E1 24063.546,E2 24063.546} C_VEL
LIN {X 0,Y 281.069,Z 899.012,A -85,B 0,C 180,E1 24070.32,E2 24070.32} C_VEL
LIN {X 0,Y 293.302,Z 869.262,A -85,B 0,C 180,E1 24076.084,E2 24076.084} C_VEL
LIN {X 0,Y 304.985,Z 836.987,A -85,B 0,C 180,E1 24080.369,E2 24080.369} C_VEL
LIN {X 0,Y 315.167,Z 801.449,A -85,B 0,C 180,E1 24083.585,E2 24083.585} C_VEL
LIN {X 0,Y 325.547,Z 754.971,A -85,B 0,C 180,E1 24086.526,E2 24086.526} C_VEL
LIN {X 0,Y 314.503,Z 684.314,A -85,B 0,C 180,E1 24096.803,E2 24096.803} C_VEL
LIN {X 0,Y 304.346,Z 666.483,A -85,B 0,C 180,E1 24103.365,E2 24103.365} C_VEL
LIN {X 0,Y 296.71,Z 654.066,A -85,B 0,C 180,E1 24110.64,E2 24110.64} C_VEL
LIN {X 0,Y 293.306,Z 647.441,A -85,B 0,C 180,E1 24117.036,E2 24117.036} C_VEL
LIN {X 0,Y 292.311,Z 646.881,A -85,B 0,C 180,E1 24120.263,E2 24120.263} C_VEL
LIN {X 0,Y 291.316,Z 650.786,A -85,B 0,C 180,E1 24123.606,E2 24123.606} C_VEL
LIN {X 0,Y 290.869,Z 656.298,A -85,B 0,C 180,E1 24126.934,E2 24126.934} C_VEL
LIN {X 0,Y 293.892,Z 663.116,A -85,B 0,C 180,E1 24133.602,E2 24133.602} C_VEL
LIN {X 0,Y 299.271,Z 673.534,A -85,B 0,C 180,E1 24139.783,E2 24139.783} C_VEL
LIN {X 0,Y 307.596,Z 691.288,A -85,B 0,C 180,E1 24146.504,E2 24146.504} C_VEL
LIN {X 0,Y 316.549,Z 712.714,A -85,B 0,C 180,E1 24152.164,E2 24152.164} C_VEL
LIN {X 0,Y 323.117,Z 735.776,A -85,B 0,C 180,E1 24156.867,E2 24156.867} C_VEL
LIN {X 0,Y 324.972,Z 748.028,A -85,B 0,C 180,E1 24159.08,E2 24159.08} C_VEL
LIN {X 0,Y 313.73,Z 782.386,A -85,B 0,C 180,E1 24162.299,E2 24162.299} C_VEL
LIN {X 0,Y 300.78,Z 813.297,A -85,B 0,C 180,E1 24166.459,E2 24166.459} C_VEL
LIN {X 0,Y 287.328,Z 840.479,A -85,B 0,C 180,E1 24171.682,E2 24171.682} C_VEL
LIN {X 0,Y 274.043,Z 864.183,A -85,B 0,C 180,E1 24178.304,E2 24178.304} C_VEL
LIN {X 0,Y 263.012,Z 882.749,A -85,B 0,C 180,E1 24186.207,E2 24186.207} C_VEL
LIN {X 0,Y 256.026,Z 894.96,A -85,B 0,C 180,E1 24194.545,E2 24194.545} C_VEL
LIN {X 0,Y 252.585,Z 901.504,A -85,B 0,C 180,E1 24203.1,E2 24203.1} C_VEL
LIN {X 0,Y 252.117,Z 903.105,A -85,B 0,C 180,E1 24209.991,E2 24209.991} C_VEL
LIN {X 0,Y 252.649,Z 901.451,A -85,B 0,C 180,E1 24216.879,E2 24216.879} C_VEL
LIN {X 0,Y 256.095,Z 894.83,A -85,B 0,C 180,E1 24225.431,E2 24225.431} C_VEL
LIN {X 0,Y 263.096,Z 882.541,A -85,B 0,C 180,E1 24233.765,E2 24233.765} C_VEL
LIN {X 0,Y 273.476,Z 865.015,A -85,B 0,C 180,E1 24241.284,E2 24241.284} C_VEL
LIN {X 0,Y 286.252,Z 842.239,A -85,B 0,C 180,E1 24247.782,E2 24247.782} C_VEL
LIN {X 0,Y 300.498,Z 813.661,A -85,B 0,C 180,E1 24253.359,E2 24253.359} C_VEL
LIN {X 0,Y 313.858,Z 781.674,A -85,B 0,C 180,E1 24257.659,E2 24257.659} C_VEL
LIN {X 0,Y 323.683,Z 750.397,A -85,B 0,C 180,E1 24260.737,E2 24260.737} C_VEL
LIN {X 0,Y 308.119,Z 764.39,A -85,B 0,C 180,E1 24262.507,E2 24262.507} C_VEL
LIN {X 0,Y 288.902,Z 779.56,A -85,B 0,C 180,E1 24265.274,E2 24265.274} C_VEL
LIN {X 0,Y 271.001,Z 791.476,A -85,B 0,C 180,E1 24268.869,E2 24268.869} C_VEL
LIN {X 0,Y 267.651,Z 793.522,A -85,B 0,C 180,E1 24270.085,E2 24270.085} C_VEL
LIN {X 0,Y 261.041,Z 828.931,A -85,B 0,C 180,E1 24275.581,E2 24275.581} C_VEL
LIN {X 0,Y 255.877,Z 858.073,A -85,B 0,C 180,E1 24281.835,E2 24281.835} C_VEL
LIN {X 0,Y 252.799,Z 881.728,A -85,B 0,C 180,E1 24288.774,E2 24288.774} C_VEL
LIN {X 0,Y 251.907,Z 898.638,A -85,B 0,C 180,E1 24295.693,E2 24295.693} C_VEL
LIN {X 0,Y 252.885,Z 911.503,A -85,B 0,C 180,E1 24303.439,E2 24303.439} C_VEL
LIN {X 0,Y 256.835,Z 918.175,A -85,B 0,C 180,E1 24310.196,E2 24310.196} C_VEL
LIN {X 0,Y 263.393,Z 920.93,A -85,B 0,C 180,E1 24316.717,E2 24316.717} C_VEL
LIN {X 0,Y 273.062,Z 920.064,A -85,B 0,C 180,E1 24322.856,E2 24322.856} C_VEL
LIN {X 0,Y 293.764,Z 912.921,A -85,B 0,C 180,E1 24331.047,E2 24331.047} C_VEL
LIN {X 0,Y 316.536,Z 902.511,A -85,B 0,C 180,E1 24336.747,E2 24336.747} C_VEL
LIN {X 0,Y 317.084,Z 902.435,A -85,B 0,C 180,E1 24337.21,E2 24337.21} C_VEL
LIN {X 0,Y 284.204,Z 927.932,A -85,B 0,C 180,E1 24346.137,E2 24346.137} C_VEL
LIN {X 0,Y 262.171,Z 948.214,A -85,B 0,C 180,E1 24357.374,E2 24357.374} C_VEL
LIN {X 0,Y 252.226,Z 961.061,A -85,B 0,C 180,E1 24368.883,E2 24368.883} C_VEL
LIN {X 0,Y 250.312,Z 965.815,A -85,B 0,C 180,E1 24375.998,E2 24375.998} C_VEL
LIN {X 0,Y 250.432,Z 967.971,A -85,B 0,C 180,E1 24383.059,E2 24383.059} C_VEL
LIN {X 0,Y 251.627,Z 967.081,A -85,B 0,C 180,E1 24390.01,E2 24390.01} C_VEL
LIN {X 0,Y 250.761,Z 963.818,A -85,B 0,C 180,E1 24398.698,E2 24398.698} C_VEL
LIN {X 0,Y 251.401,Z 955.63,A -85,B 0,C 180,E1 24407.549,E2 24407.549} C_VEL
LIN {X 0,Y 255.251,Z 942.195,A -85,B 0,C 180,E1 24416.107,E2 24416.107} C_VEL
LIN {X 0,Y 263.216,Z 923.109,A -85,B 0,C 180,E1 24424.182,E2 24424.182} C_VEL
LIN {X 0,Y 274.014,Z 899.396,A -85,B 0,C 180,E1 24431.056,E2 24431.056} C_VEL
LIN {X 0,Y 286.259,Z 871.22,A -85,B 0,C 180,E1 24436.735,E2 24436.735} C_VEL
LIN {X 0,Y 298.743,Z 838.62,A -85,B 0,C 180,E1 24441.256,E2 24441.256} C_VEL
LIN {X 0,Y 309.495,Z 803.406,A -85,B 0,C 180,E1 24444.552,E2 24444.552} C_VEL
LIN {X 0,Y 320.092,Z 757.001,A -85,B 0,C 180,E1 24447.594,E2 24447.594} C_VEL
LIN {X 0,Y 311.021,Z 690.989,A -85,B 0,C 180,E1 24457.42,E2 24457.42} C_VEL
LIN {X 0,Y 302.056,Z 673.946,A -85,B 0,C 180,E1 24463.61,E2 24463.61} C_VEL
LIN {X 0,Y 294.657,Z 661.604,A -85,B 0,C 180,E1 24470.926,E2 24470.926} C_VEL
LIN {X 0,Y 291.176,Z 654.996,A -85,B 0,C 180,E1 24477.793,E2 24477.793} C_VEL
LIN {X 0,Y 290.869,Z 655.719,A -85,B 0,C 180,E1 24486.539,E2 24486.539} C_VEL
LIN {X 0,Y 290.869,Z 656.298,A -85,B 0,C 180,E1 24486.934,E2 24486.934} C_VEL
LIN {X 0,Y 290.963,Z 662.801,A -85,B 0,C 180,E1 24490.122,E2 24490.122} C_VEL
LIN {X 0,Y 291.533,Z 670.433,A -85,B 0,C 180,E1 24493.248,E2 24493.248} C_VEL
LIN {X 0,Y 296.571,Z 680.705,A -85,B 0,C 180,E1 24499.387,E2 24499.387} C_VEL
LIN {X 0,Y 304.391,Z 698.049,A -85,B 0,C 180,E1 24506.025,E2 24506.025} C_VEL
LIN {X 0,Y 312.867,Z 719.517,A -85,B 0,C 180,E1 24511.769,E2 24511.769} C_VEL
LIN {X 0,Y 318.51,Z 742.88,A -85,B 0,C 180,E1 24516.639,E2 24516.639} C_VEL
LIN {X 0,Y 319.297,Z 751.86,A -85,B 0,C 180,E1 24518.217,E2 24518.217} C_VEL
LIN {X 0,Y 307.279,Z 786.444,A -85,B 0,C 180,E1 24521.567,E2 24521.567} C_VEL
LIN {X 0,Y 293.711,Z 817.475,A -85,B 0,C 180,E1 24525.916,E2 24525.916} C_VEL
LIN {X 0,Y 279.089,Z 845.254,A -85,B 0,C 180,E1 24531.582,E2 24531.582} C_VEL
LIN {X 0,Y 266.038,Z 867.386,A -85,B 0,C 180,E1 24538.198,E2 24538.198} C_VEL
LIN {X 0,Y 255.828,Z 883.762,A -85,B 0,C 180,E1 24545.496,E2 24545.496} C_VEL
LIN {X 0,Y 248.442,Z 895.967,A -85,B 0,C 180,E1 24554.061,E2 24554.061} C_VEL
LIN {X 0,Y 244.795,Z 902.498,A -85,B 0,C 180,E1 24562.879,E2 24562.879} C_VEL
LIN {X 0,Y 244.293,Z 904.091,A -85,B 0,C 180,E1 24569.99,E2 24569.99} C_VEL
LIN {X 0,Y 245.227,Z 901.604,A -85,B 0,C 180,E1 24578.768,E2 24578.768} C_VEL
LIN {X 0,Y 249.696,Z 893.811,A -85,B 0,C 180,E1 24587.652,E2 24587.652} C_VEL
LIN {X 0,Y 257.906,Z 880.407,A -85,B 0,C 180,E1 24596.134,E2 24596.134} C_VEL
LIN {X 0,Y 269.586,Z 861.465,A -85,B 0,C 180,E1 24603.702,E2 24603.702} C_VEL
LIN {X 0,Y 282.997,Z 838.047,A -85,B 0,C 180,E1 24609.967,E2 24609.967} C_VEL
LIN {X 0,Y 296.958,Z 810.272,A -85,B 0,C 180,E1 24615.112,E2 24615.112} C_VEL
LIN {X 0,Y 310.232,Z 778.486,A -85,B 0,C 180,E1 24619.192,E2 24619.192} C_VEL
LIN {X 0,Y 314.516,Z 766.35,A -85,B 0,C 180,E1 24620.415,E2 24620.415} C_VEL
LIN {X 0,Y 313.948,Z 765.382,A -85,B 0,C 180,E1 24620.743,E2 24620.743} C_VEL
LIN {X 0,Y 289.525,Z 784.079,A -85,B 0,C 180,E1 24623.945,E2 24623.945} C_VEL
LIN {X 0,Y 269.46,Z 797.017,A -85,B 0,C 180,E1 24627.725,E2 24627.725} C_VEL
LIN {X 0,Y 258.678,Z 802.721,A -85,B 0,C 180,E1 24630.634,E2 24630.634} C_VEL
LIN {X 0,Y 250.654,Z 843.202,A -85,B 0,C 180,E1 24638.045,E2 24638.045} C_VEL
LIN {X 0,Y 246.309,Z 870.108,A -85,B 0,C 180,E1 24644.852,E2 24644.852} C_VEL
LIN {X 0,Y 244.177,Z 891.646,A -85,B 0,C 180,E1 24652.429,E2 24652.429} C_VEL
LIN {X 0,Y 244.289,Z 906.738,A -85,B 0,C 180,E1 24660.004,E2 24660.004} C_VEL
LIN {X 0,Y 246.767,Z 916.008,A -85,B 0,C 180,E1 24667.057,E2 24667.057} C_VEL
LIN {X 0,Y 252.134,Z 921.106,A -85,B 0,C 180,E1 24673.91,E2 24673.91} C_VEL
LIN {X 0,Y 260.623,Z 922.54,A -85,B 0,C 180,E1 24680.415,E2 24680.415} C_VEL
LIN {X 0,Y 279.511,Z 918.551,A -85,B 0,C 180,E1 24689.199,E2 24689.199} C_VEL
LIN {X 0,Y 307.233,Z 907.874,A -85,B 0,C 180,E1 24696.797,E2 24696.797} C_VEL
LIN {X 0,Y 303.178,Z 910.957,A -85,B 0,C 180,E1 24698.093,E2 24698.093} C_VEL
LIN {X 0,Y 272.744,Z 933.046,A -85,B 0,C 180,E1 24707.141,E2 24707.141} C_VEL
LIN {X 0,Y 251.709,Z 951.54,A -85,B 0,C 180,E1 24719.236,E2 24719.236} C_VEL
LIN {X 0,Y 243.8,Z 961.651,A -85,B 0,C 180,E1 24730.092,E2 24730.092} C_VEL
LIN {X 0,Y 242.354,Z 966.006,A -85,B 0,C 180,E1 24739.2,E2 24739.2} C_VEL
LIN {X 0,Y 243.201,Z 966.516,A -85,B 0,C 180,E1 24746.438,E2 24746.438} C_VEL
LIN {X 0,Y 243.85,Z 965.63,A -85,B 0,C 180,E1 24750.01,E2 24750.01} C_VEL
LIN {X 0,Y 243.045,Z 963.818,A -85,B 0,C 180,E1 24757.172,E2 24757.172} C_VEL
LIN {X 0,Y 243.137,Z 957.468,A -85,B 0,C 180,E1 24765.517,E2 24765.517} C_VEL
LIN {X 0,Y 246.232,Z 945.51,A -85,B 0,C 180,E1 24774.456,E2 24774.456} C_VEL
LIN {X 0,Y 253.624,Z 927.878,A -85,B 0,C 180,E1 24782.999,E2 24782.999} C_VEL
LIN {X 0,Y 264.788,Z 904.447,A -85,B 0,C 180,E1 24790.623,E2 24790.623} C_VEL
LIN {X 0,Y 277.673,Z 876.848,A -85,B 0,C 180,E1 24796.754,E2 24796.754} C_VEL
LIN {X 0,Y 290.51,Z 845.831,A -85,B 0,C 180,E1 24801.49,E2 24801.49} C_VEL
LIN {X 0,Y 302.293,Z 811.137,A -85,B 0,C 180,E1 24805.075,E2 24805.075} C_VEL
LIN {X 0,Y 314.231,Z 763.627,A -85,B 0,C 180,E1 24808.336,E2 24808.336} C_VEL
LIN {X 0,Y 314.56,Z 757.85,A -85,B 0,C 180,E1 24808.906,E2 24808.906} C_VEL
LIN {X 0,Y 307.015,Z 695.489,A -85,B 0,C 180,E1 24818.547,E2 24818.547} C_VEL
LIN {X 0,Y 298.744,Z 680.186,A -85,B 0,C 180,E1 24824.586,E2 24824.586} C_VEL
LIN {X 0,Y 292.529,Z 669.075,A -85,B 0,C 180,E1 24831.246,E2 24831.246} C_VEL
LIN {X 0,Y 289.423,Z 662.668,A -85,B 0,C 180,E1 24837.779,E2 24837.779} C_VEL
LIN {X 0,Y 288.892,Z 663.344,A -85,B 0,C 180,E1 24846.3,E2 24846.3} C_VEL
LIN {X 0,Y 291.533,Z 670.433,A -85,B 0,C 180,E1 24853.248,E2 24853.248} C_VEL
LIN {X 0,Y 292.683,Z 678.92,A -85,B 0,C 180,E1 24856.247,E2 24856.247} C_VEL
LIN {X 0,Y 294.019,Z 688.325,A -85,B 0,C 180,E1 24859.163,E2 24859.163} C_VEL
LIN {X 0,Y 301.341,Z 705.227,A -85,B 0,C 180,E1 24865.682,E2 24865.682} C_VEL
LIN {X 0,Y 309.115,Z 726.868,A -85,B 0,C 180,E1 24871.516,E2 24871.516} C_VEL
LIN {X 0,Y 313.626,Z 748.777,A -85,B 0,C 180,E1 24876.172,E2 24876.172} C_VEL
LIN {X 0,Y 313.68,Z 755.638,A -85,B 0,C 180,E1 24877.309,E2 24877.309} C_VEL
LIN {X 0,Y 300.688,Z 791.092,A -85,B 0,C 180,E1 24880.886,E2 24880.886} C_VEL
LIN {X 0,Y 286.501,Z 821.666,A -85,B 0,C 180,E1 24885.386,E2 24885.386} C_VEL
LIN {X 0,Y 272.189,Z 847.7,A -85,B 0,C 180,E1 24890.902,E2 24890.902} C_VEL
LIN {X 0,Y 258.68,Z 869.473,A -85,B 0,C 180,E1 24897.68,E2 24897.68} C_VEL
LIN {X 0,Y 247.646,Z 886.461,A -85,B 0,C 180,E1 24905.693,E2 24905.693} C_VEL
LIN {X 0,Y 240.879,Z 896.974,A -85,B 0,C 180,E1 24913.547,E2 24913.547} C_VEL
LIN {X 0,Y 237.002,Z 903.488,A -85,B 0,C 180,E1 24922.644,E2 24922.644} C_VEL
LIN {X 0,Y 236.466,Z 905.078,A -85,B 0,C 180,E1 24929.99,E2 24929.99} C_VEL
LIN {X 0,Y 237.063,Z 903.437,A -85,B 0,C 180,E1 24937.334,E2 24937.334} C_VEL
LIN {X 0,Y 240.957,Z 896.841,A -85,B 0,C 180,E1 24946.427,E2 24946.427} C_VEL
LIN {X 0,Y 248.753,Z 884.598,A -85,B 0,C 180,E1 24955.228,E2 24955.228} C_VEL
LIN {X 0,Y 260.869,Z 865.95,A -85,B 0,C 180,E1 24963.479,E2 24963.479} C_VEL
LIN {X 0,Y 274.337,Z 843.774,A -85,B 0,C 180,E1 24969.933,E2 24969.933} C_VEL
LIN {X 0,Y 289.367,Z 815.694,A -85,B 0,C 180,E1 24975.506,E2 24975.506} C_VEL
LIN {X 0,Y 303.48,Z 783.928,A -85,B 0,C 180,E1 24979.832,E2 24979.832} C_VEL
LIN {X 0,Y 305.162,Z 779.576,A -85,B 0,C 180,E1 24980.305,E2 24980.305} C_VEL
LIN {X 0,Y 305.007,Z 777.841,A -85,B 0,C 180,E1 24980.714,E2 24980.714} C_VEL
LIN {X 0,Y 286.085,Z 791.221,A -85,B 0,C 180,E1 24983.25,E2 24983.25} C_VEL
LIN {X 0,Y 265.367,Z 803.726,A -85,B 0,C 180,E1 24987.165,E2 24987.165} C_VEL
LIN {X 0,Y 250.372,Z 811.919,A -85,B 0,C 180,E1 24991.055,E2 24991.055} C_VEL
LIN {X 0,Y 248.879,Z 812.685,A -85,B 0,C 180,E1 24991.849,E2 24991.849} C_VEL
LIN {X 0,Y 242.323,Z 846.462,A -85,B 0,C 180,E1 24998.401,E2 24998.401} C_VEL
LIN {X 0,Y 237.99,Z 873.591,A -85,B 0,C 180,E1 25005.725,E2 25005.725} C_VEL
LIN {X 0,Y 236.153,Z 894.694,A -85,B 0,C 180,E1 25013.671,E2 25013.671} C_VEL
LIN {X 0,Y 236.515,Z 908.279,A -85,B 0,C 180,E1 25020.922,E2 25020.922} C_VEL
LIN {X 0,Y 240.098,Z 918.294,A -85,B 0,C 180,E1 25029.08,E2 25029.08} C_VEL
LIN {X 0,Y 248.532,Z 923.533,A -85,B 0,C 180,E1 25037.749,E2 25037.749} C_VEL
LIN {X 0,Y 259.03,Z 923.847,A -85,B 0,C 180,E1 25044.17,E2 25044.17} C_VEL
LIN {X 0,Y 281.2,Z 918.57,A -85,B 0,C 180,E1 25052.601,E2 25052.601} C_VEL
LIN {X 0,Y 296.89,Z 913.167,A -85,B 0,C 180,E1 25056.626,E2 25056.626} C_VEL
LIN {X 0,Y 297.609,Z 913.092,A -85,B 0,C 180,E1 25057.101,E2 25057.101} C_VEL
LIN {X 0,Y 265.037,Z 934.856,A -85,B 0,C 180,E1 25066.695,E2 25066.695} C_VEL
LIN {X 0,Y 244.681,Z 951.157,A -85,B 0,C 180,E1 25078.251,E2 25078.251} C_VEL
LIN {X 0,Y 235.498,Z 961.784,A -85,B 0,C 180,E1 25091.245,E2 25091.245} C_VEL
LIN {X 0,Y 234.507,Z 964.752,A -85,B 0,C 180,E1 25098.834,E2 25098.834} C_VEL
LIN {X 0,Y 235.397,Z 965.027,A -85,B 0,C 180,E1 25106.32,E2 25106.32} C_VEL
LIN {X 0,Y 236.013,Z 964.642,A -85,B 0,C 180,E1 25110.01,E2 25110.01} C_VEL
LIN {X 0,Y 235.162,Z 962.812,A -85,B 0,C 180,E1 25117.414,E2 25117.414} C_VEL
LIN {X 0,Y 235.474,Z 955.633,A -85,B 0,C 180,E1 25126.842,E2 25126.842} C_VEL
LIN {X 0,Y 239.393,Z 942.721,A -85,B 0,C 180,E1 25136.31,E2 25136.31} C_VEL
LIN {X 0,Y 247.768,Z 924.5,A -85,B 0,C 180,E1 25144.945,E2 25144.945} C_VEL
LIN {X 0,Y 259.308,Z 901.747,A -85,B 0,C 180,E1 25152.232,E2 25152.232} C_VEL
LIN {X 0,Y 272.924,Z 873.623,A -85,B 0,C 180,E1 25158.404,E2 25158.404} C_VEL
LIN {X 0,Y 286.505,Z 841.803,A -85,B 0,C 180,E1 25163.134,E2 25163.134} C_VEL
LIN {X 0,Y 298.566,Z 806.931,A -85,B 0,C 180,E1 25166.612,E2 25166.612} C_VEL
LIN {X 0,Y 309.68,Z 763.885,A -85,B 0,C 180,E1 25169.52,E2 25169.52} C_VEL
LIN {X 0,Y 303.594,Z 701.857,A -85,B 0,C 180,E1 25179.171,E2 25179.171} C_VEL
LIN {X 0,Y 295.909,Z 686.853,A -85,B 0,C 180,E1 25185.26,E2 25185.26} C_VEL
LIN {X 0,Y 290.104,Z 676.279,A -85,B 0,C 180,E1 25191.929,E2 25191.929} C_VEL
LIN {X 0,Y 287.549,Z 670.315,A -85,B 0,C 180,E1 25197.765,E2 25197.765} C_VEL
LIN {X 0,Y 286.93,Z 671.046,A -85,B 0,C 180,E1 25206.153,E2 25206.153} C_VEL
LIN {X 0,Y 289.385,Z 678.24,A -85,B 0,C 180,E1 25213.139,E2 25213.139} C_VEL
LIN {X 0,Y 293.795,Z 687.673,A -85,B 0,C 180,E1 25218.89,E2 25218.89} C_VEL
LIN {X 0,Y 294.019,Z 688.325,A -85,B 0,C 180,E1 25219.163,E2 25219.163} C_VEL
LIN {X 0,Y 295.544,Z 698.729,A -85,B 0,C 180,E1 25221.892,E2 25221.892} C_VEL
LIN {X 0,Y 297.269,Z 709.931,A -85,B 0,C 180,E1 25224.524,E2 25224.524} C_VEL
LIN {X 0,Y 304.541,Z 731.168,A -85,B 0,C 180,E1 25230.546,E2 25230.546} C_VEL
LIN {X 0,Y 308.547,Z 753.543,A -85,B 0,C 180,E1 25235.492,E2 25235.492} C_VEL
LIN {X 0,Y 308.206,Z 759.094,A -85,B 0,C 180,E1 25236.362,E2 25236.362} C_VEL
LIN {X 0,Y 294.879,Z 793.935,A -85,B 0,C 180,E1 25239.957,E2 25239.957} C_VEL
LIN {X 0,Y 280.364,Z 823.863,A -85,B 0,C 180,E1 25244.466,E2 25244.466} C_VEL
LIN {X 0,Y 265.609,Z 849.65,A -85,B 0,C 180,E1 25250.064,E2 25250.064} C_VEL
LIN {X 0,Y 251.352,Z 871.555,A -85,B 0,C 180,E1 25257.132,E2 25257.132} C_VEL
LIN {X 0,Y 239.625,Z 888.724,A -85,B 0,C 180,E1 25265.721,E2 25265.721} C_VEL
LIN {X 0,Y 232.184,Z 899.664,A -85,B 0,C 180,E1 25274.858,E2 25274.858} C_VEL
LIN {X 0,Y 229.23,Z 904.48,A -85,B 0,C 180,E1 25282.393,E2 25282.393} C_VEL
LIN {X 0,Y 228.642,Z 906.064,A -85,B 0,C 180,E1 25289.99,E2 25289.99} C_VEL
LIN {X 0,Y 229.322,Z 904.356,A -85,B 0,C 180,E1 25297.776,E2 25297.776} C_VEL
LIN {X 0,Y 233.423,Z 897.846,A -85,B 0,C 180,E1 25306.973,E2 25306.973} C_VEL
LIN {X 0,Y 241.652,Z 885.616,A -85,B 0,C 180,E1 25316.024,E2 25316.024} C_VEL
LIN {X 0,Y 253.597,Z 868.133,A -85,B 0,C 180,E1 25324.054,E2 25324.054} C_VEL
LIN {X 0,Y 268.371,Z 844.842,A -85,B 0,C 180,E1 25331.01,E2 25331.01} C_VEL
LIN {X 0,Y 283.925,Z 816.777,A -85,B 0,C 180,E1 25336.631,E2 25336.631} C_VEL
LIN {X 0,Y 296.52,Z 789.091,A -85,B 0,C 180,E1 25340.576,E2 25340.576} C_VEL
LIN {X 0,Y 272.236,Z 804.252,A -85,B 0,C 180,E1 25344.253,E2 25344.253} C_VEL
LIN {X 0,Y 250.432,Z 816.142,A -85,B 0,C 180,E1 25349.116,E2 25349.116} C_VEL
LIN {X 0,Y 239.709,Z 821.022,A -85,B 0,C 180,E1 25352.712,E2 25352.712} C_VEL
LIN {X 0,Y 233.176,Z 854.093,A -85,B 0,C 180,E1 25359.911,E2 25359.911} C_VEL
LIN {X 0,Y 229.408,Z 879.7,A -85,B 0,C 180,E1 25367.612,E2 25367.612} C_VEL
LIN {X 0,Y 228.23,Z 898.443,A -85,B 0,C 180,E1 25375.411,E2 25375.411} C_VEL
LIN {X 0,Y 229.257,Z 912.506,A -85,B 0,C 180,E1 25383.794,E2 25383.794} C_VEL
LIN {X 0,Y 235.22,Z 921.923,A -85,B 0,C 180,E1 25393.032,E2 25393.032} C_VEL
LIN {X 0,Y 246.152,Z 925.544,A -85,B 0,C 180,E1 25401.674,E2 25401.674} C_VEL
LIN {X 0,Y 266.501,Z 923.426,A -85,B 0,C 180,E1 25410.775,E2 25410.775} C_VEL
LIN {X 0,Y 287.702,Z 917.54,A -85,B 0,C 180,E1 25416.702,E2 25416.702} C_VEL
LIN {X 0,Y 278.104,Z 923.455,A -85,B 0,C 180,E1 25419.364,E2 25419.364} C_VEL
LIN {X 0,Y 245.532,Z 944.633,A -85,B 0,C 180,E1 25431.907,E2 25431.907} C_VEL
LIN {X 0,Y 230.714,Z 957.177,A -85,B 0,C 180,E1 25444.741,E2 25444.741} C_VEL
LIN {X 0,Y 226.949,Z 962.462,A -85,B 0,C 180,E1 25454.522,E2 25454.522} C_VEL
LIN {X 0,Y 226.926,Z 963.86,A -85,B 0,C 180,E1 25462.336,E2 25462.336} C_VEL
LIN {X 0,Y 228.172,Z 963.654,A -85,B 0,C 180,E1 25470.01,E2 25470.01} C_VEL
LIN {X 0,Y 227.288,Z 961.806,A -85,B 0,C 180,E1 25477.673,E2 25477.673} C_VEL
LIN {X 0,Y 227.7,Z 954.578,A -85,B 0,C 180,E1 25487.435,E2 25487.435} C_VEL
LIN {X 0,Y 232.042,Z 941.618,A -85,B 0,C 180,E1 25497.211,E2 25497.211} C_VEL
LIN {X 0,Y 241.084,Z 923.244,A -85,B 0,C 180,E1 25506.114,E2 25506.114} C_VEL
LIN {X 0,Y 253.364,Z 900.24,A -85,B 0,C 180,E1 25513.589,E2 25513.589} C_VEL
LIN {X 0,Y 267.895,Z 871.562,A -85,B 0,C 180,E1 25519.88,E2 25519.88} C_VEL
LIN {X 0,Y 282.165,Z 839.322,A -85,B 0,C 180,E1 25524.616,E2 25524.616} C_VEL
LIN {X 0,Y 294.613,Z 804.116,A -85,B 0,C 180,E1 25528.075,E2 25528.075} C_VEL
LIN {X 0,Y 304.72,Z 765.566,A -85,B 0,C 180,E1 25530.701,E2 25530.701} C_VEL
LIN {X 0,Y 299.895,Z 707.517,A -85,B 0,C 180,E1 25540.06,E2 25540.06} C_VEL
LIN {X 0,Y 292.92,Z 693.439,A -85,B 0,C 180,E1 25545.967,E2 25545.967} C_VEL
LIN {X 0,Y 287.697,Z 683.543,A -85,B 0,C 180,E1 25552.432,E2 25552.432} C_VEL
LIN {X 0,Y 285.317,Z 677.828,A -85,B 0,C 180,E1 25558.475,E2 25558.475} C_VEL
LIN {X 0,Y 284.883,Z 678.712,A -85,B 0,C 180,E1 25566.005,E2 25566.005} C_VEL
LIN {X 0,Y 287.121,Z 685.687,A -85,B 0,C 180,E1 25572.857,E2 25572.857} C_VEL
LIN {X 0,Y 291.32,Z 695.36,A -85,B 0,C 180,E1 25578.704,E2 25578.704} C_VEL
LIN {X 0,Y 297.269,Z 709.931,A -85,B 0,C 180,E1 25584.524,E2 25584.524} C_VEL
LIN {X 0,Y 298.773,Z 721.939,A -85,B 0,C 180,E1 25586.962,E2 25586.962} C_VEL
LIN {X 0,Y 299.78,Z 734.66,A -85,B 0,C 180,E1 25589.322,E2 25589.322} C_VEL
LIN {X 0,Y 303.242,Z 755.498,A -85,B 0,C 180,E1 25594.199,E2 25594.199} C_VEL
LIN {X 0,Y 303.237,Z 761.271,A -85,B 0,C 180,E1 25595.272,E2 25595.272} C_VEL
LIN {X 0,Y 289.454,Z 796.051,A -85,B 0,C 180,E1 25598.9,E2 25598.9} C_VEL
LIN {X 0,Y 273.857,Z 826.882,A -85,B 0,C 180,E1 25603.658,E2 25603.658} C_VEL
LIN {X 0,Y 257.791,Z 853.447,A -85,B 0,C 180,E1 25609.707,E2 25609.707} C_VEL
LIN {X 0,Y 243.065,Z 875.086,A -85,B 0,C 180,E1 25617.151,E2 25617.151} C_VEL
LIN {X 0,Y 231.477,Z 891.082,A -85,B 0,C 180,E1 25625.84,E2 25625.84} C_VEL
LIN {X 0,Y 224.594,Z 900.67,A -85,B 0,C 180,E1 25634.333,E2 25634.333} C_VEL
LIN {X 0,Y 221.452,Z 905.474,A -85,B 0,C 180,E1 25642.124,E2 25642.124} C_VEL
LIN {X 0,Y 220.822,Z 907.05,A -85,B 0,C 180,E1 25649.989,E2 25649.989} C_VEL
LIN {X 0,Y 221.506,Z 905.425,A -85,B 0,C 180,E1 25657.852,E2 25657.852} C_VEL
LIN {X 0,Y 225.906,Z 898.85,A -85,B 0,C 180,E1 25667.556,E2 25667.556} C_VEL
LIN {X 0,Y 234.602,Z 886.641,A -85,B 0,C 180,E1 25676.867,E2 25676.867} C_VEL
LIN {X 0,Y 247.13,Z 869.171,A -85,B 0,C 180,E1 25685.074,E2 25685.074} C_VEL
LIN {X 0,Y 262.506,Z 845.913,A -85,B 0,C 180,E1 25692.132,E2 25692.132} C_VEL
LIN {X 0,Y 278.615,Z 817.83,A -85,B 0,C 180,E1 25697.802,E2 25697.802} C_VEL
LIN {X 0,Y 286.371,Z 802.198,A -85,B 0,C 180,E1 25700.165,E2 25700.165} C_VEL
LIN {X 0,Y 286.449,Z 800.49,A -85,B 0,C 180,E1 25700.613,E2 25700.613} C_VEL
LIN {X 0,Y 261.979,Z 814.29,A -85,B 0,C 180,E1 25704.678,E2 25704.678} C_VEL
LIN {X 0,Y 238.608,Z 825.918,A -85,B 0,C 180,E1 25710.625,E2 25710.625} C_VEL
LIN {X 0,Y 230.556,Z 829.442,A -85,B 0,C 180,E1 25713.677,E2 25713.677} C_VEL
LIN {X 0,Y 223.622,Z 864.521,A -85,B 0,C 180,E1 25722.491,E2 25722.491} C_VEL
LIN {X 0,Y 220.76,Z 887.851,A -85,B 0,C 180,E1 25730.625,E2 25730.625} C_VEL
LIN {X 0,Y 220.535,Z 905.141,A -85,B 0,C 180,E1 25739.021,E2 25739.021} C_VEL
LIN {X 0,Y 223.324,Z 917.452,A -85,B 0,C 180,E1 25747.802,E2 25747.802} C_VEL
LIN {X 0,Y 229.409,Z 923.974,A -85,B 0,C 180,E1 25755.321,E2 25755.321} C_VEL
LIN {X 0,Y 238.953,Z 926.993,A -85,B 0,C 180,E1 25762.362,E2 25762.362} C_VEL
LIN {X 0,Y 260.024,Z 925.669,A -85,B 0,C 180,E1 25771.628,E2 25771.628} C_VEL
LIN {X 0,Y 278.37,Z 921.57,A -85,B 0,C 180,E1 25776.776,E2 25776.776} C_VEL
LIN {X 0,Y 244.356,Z 941.168,A -85,B 0,C 180,E1 25788.075,E2 25788.075} C_VEL
LIN {X 0,Y 224.799,Z 954.916,A -85,B 0,C 180,E1 25801.86,E2 25801.86} C_VEL
LIN {X 0,Y 219.177,Z 961.19,A -85,B 0,C 180,E1 25813.958,E2 25813.958} C_VEL
LIN {X 0,Y 219.108,Z 962.461,A -85,B 0,C 180,E1 25822.061,E2 25822.061} C_VEL
LIN {X 0,Y 220.315,Z 962.663,A -85,B 0,C 180,E1 25830.011,E2 25830.011} C_VEL
LIN {X 0,Y 219.406,Z 960.798,A -85,B 0,C 180,E1 25837.95,E2 25837.95} C_VEL
LIN {X 0,Y 219.578,Z 955.438,A -85,B 0,C 180,E1 25846.034,E2 25846.034} C_VEL
LIN {X 0,Y 223.337,Z 943.63,A -85,B 0,C 180,E1 25856.179,E2 25856.179} C_VEL
LIN {X 0,Y 232.512,Z 925.47,A -85,B 0,C 180,E1 25865.922,E2 25865.922} C_VEL
LIN {X 0,Y 245.816,Z 901.902,A -85,B 0,C 180,E1 25874.13,E2 25874.13} C_VEL
LIN {X 0,Y 260.2,Z 875.124,A -85,B 0,C 180,E1 25880.39,E2 25880.39} C_VEL
LIN {X 0,Y 275.214,Z 843.435,A -85,B 0,C 180,E1 25885.355,E2 25885.355} C_VEL
LIN {X 0,Y 288.524,Z 808.743,A -85,B 0,C 180,E1 25888.96,E2 25888.96} C_VEL
LIN {X 0,Y 299.723,Z 768.264,A -85,B 0,C 180,E1 25891.815,E2 25891.815} C_VEL
LIN {X 0,Y 296.242,Z 713.07,A -85,B 0,C 180,E1 25900.97,E2 25900.97} C_VEL
LIN {X 0,Y 289.347,Z 698.558,A -85,B 0,C 180,E1 25907.428,E2 25907.428} C_VEL
LIN {X 0,Y 285.318,Z 690.814,A -85,B 0,C 180,E1 25912.943,E2 25912.943} C_VEL
LIN {X 0,Y 283.398,Z 685.478,A -85,B 0,C 180,E1 25918.465,E2 25918.465} C_VEL
LIN {X 0,Y 282.768,Z 686.25,A -85,B 0,C 180,E1 25925.761,E2 25925.761} C_VEL
LIN {X 0,Y 284.696,Z 693.288,A -85,B 0,C 180,E1 25932.682,E2 25932.682} C_VEL
LIN {X 0,Y 288.667,Z 702.817,A -85,B 0,C 180,E1 25938.438,E2 25938.438} C_VEL
LIN {X 0,Y 295.009,Z 719.101,A -85,B 0,C 180,E1 25944.858,E2 25944.858} C_VEL
LIN {X 0,Y 299.78,Z 734.66,A -85,B 0,C 180,E1 25949.322,E2 25949.322} C_VEL
LIN {X 0,Y 300.082,Z 744.213,A -85,B 0,C 180,E1 25951.041,E2 25951.041} C_VEL
LIN {X 0,Y 298.368,Z 761.437,A -85,B 0,C 180,E1 25953.718,E2 25953.718} C_VEL
LIN {X 0,Y 297.423,Z 766.016,A -85,B 0,C 180,E1 25954.37,E2 25954.37} C_VEL
LIN {X 0,Y 283.185,Z 800.057,A -85,B 0,C 180,E1 25958.056,E2 25958.056} C_VEL
LIN {X 0,Y 266.998,Z 830.639,A -85,B 0,C 180,E1 25962.953,E2 25962.953} C_VEL
LIN {X 0,Y 250.205,Z 856.922,A -85,B 0,C 180,E1 25969.251,E2 25969.251} C_VEL
LIN {X 0,Y 235.32,Z 877.617,A -85,B 0,C 180,E1 25976.803,E2 25976.803} C_VEL
LIN {X 0,Y 223.329,Z 893.431,A -85,B 0,C 180,E1 25985.967,E2 25985.967} C_VEL
LIN {X 0,Y 215.948,Z 903.182,A -85,B 0,C 180,E1 25995.773,E2 25995.773} C_VEL
LIN {X 0,Y 212.998,Z 907.639,A -85,B 0,C 180,E1 26005.909,E2 26005.909} C_VEL
LIN {X 0,Y 213.098,Z 907.599,A -85,B 0,C 180,E1 26014.066,E2 26014.066} C_VEL
LIN {X 0,Y 216.027,Z 903.091,A -85,B 0,C 180,E1 26024.199,E2 26024.199} C_VEL
LIN {X 0,Y 223.414,Z 893.26,A -85,B 0,C 180,E1 26034,E2 26034} C_VEL
LIN {X 0,Y 235.554,Z 877.143,A -85,B 0,C 180,E1 26043.283,E2 26043.283} C_VEL
LIN {X 0,Y 250.64,Z 856.07,A -85,B 0,C 180,E1 26050.867,E2 26050.867} C_VEL
LIN {X 0,Y 267.194,Z 829.91,A -85,B 0,C 180,E1 26057.066,E2 26057.066} C_VEL
LIN {X 0,Y 277.8,Z 809.972,A -85,B 0,C 180,E1 26060.527,E2 26060.527} C_VEL
LIN {X 0,Y 251.49,Z 823.725,A -85,B 0,C 180,E1 26065.224,E2 26065.224} C_VEL
LIN {X 0,Y 227.426,Z 834.752,A -85,B 0,C 180,E1 26072.213,E2 26072.213} C_VEL
LIN {X 0,Y 220.914,Z 837.4,A -85,B 0,C 180,E1 26075.17,E2 26075.17} C_VEL
LIN {X 0,Y 215.495,Z 866.429,A -85,B 0,C 180,E1 26082.845,E2 26082.845} C_VEL
LIN {X 0,Y 212.723,Z 889.561,A -85,B 0,C 180,E1 26091.301,E2 26091.301} C_VEL
LIN {X 0,Y 212.715,Z 906.665,A -85,B 0,C 180,E1 26100.005,E2 26100.005} C_VEL
LIN {X 0,Y 216.815,Z 919.835,A -85,B 0,C 180,E1 26110.065,E2 26110.065} C_VEL
LIN {X 0,Y 226.367,Z 926.945,A -85,B 0,C 180,E1 26119.554,E2 26119.554} C_VEL
LIN {X 0,Y 238.119,Z 928.918,A -85,B 0,C 180,E1 26126.45,E2 26126.45} C_VEL
LIN {X 0,Y 262.646,Z 926.424,A -85,B 0,C 180,E1 26135.229,E2 26135.229} C_VEL
LIN {X 0,Y 267.219,Z 925.566,A -85,B 0,C 180,E1 26136.448,E2 26136.448} C_VEL
LIN {X 0,Y 266.377,Z 926.318,A -85,B 0,C 180,E1 26137.232,E2 26137.232} C_VEL
LIN {X 0,Y 232.88,Z 944.218,A -85,B 0,C 180,E1 26149.424,E2 26149.424} C_VEL
LIN {X 0,Y 214.626,Z 956.555,A -85,B 0,C 180,E1 26164.951,E2 26164.951} C_VEL
LIN {X 0,Y 211.074,Z 960.709,A -85,B 0,C 180,E1 26177.575,E2 26177.575} C_VEL
LIN {X 0,Y 212.169,Z 961.544,A -85,B 0,C 180,E1 26188.566,E2 26188.566} C_VEL
LIN {X 0,Y 211.888,Z 961.125,A -85,B 0,C 180,E1 26194.112,E2 26194.112} C_VEL
LIN {X 0,Y 211.416,Z 957.495,A -85,B 0,C 180,E1 26202.428,E2 26202.428} C_VEL
LIN {X 0,Y 213.537,Z 948.239,A -85,B 0,C 180,E1 26212.73,E2 26212.73} C_VEL
LIN {X 0,Y 221.224,Z 932.424,A -85,B 0,C 180,E1 26223.238,E2 26223.238} C_VEL
LIN {X 0,Y 233.048,Z 912.139,A -85,B 0,C 180,E1 26231.915,E2 26231.915} C_VEL
LIN {X 0,Y 247.999,Z 886.637,A -85,B 0,C 180,E1 26239.134,E2 26239.134} C_VEL
LIN {X 0,Y 263.457,Z 857.547,A -85,B 0,C 180,E1 26244.623,E2 26244.623} C_VEL
LIN {X 0,Y 278.18,Z 824.359,A -85,B 0,C 180,E1 26248.806,E2 26248.806} C_VEL
LIN {X 0,Y 290.623,Z 787.142,A -85,B 0,C 180,E1 26251.919,E2 26251.919} C_VEL
LIN {X 0,Y 294.895,Z 770.786,A -85,B 0,C 180,E1 26253.01,E2 26253.01} C_VEL
LIN {X 0,Y 292.626,Z 718.814,A -85,B 0,C 180,E1 26261.808,E2 26261.808} C_VEL
LIN {X 0,Y 286.196,Z 704.583,A -85,B 0,C 180,E1 26268.451,E2 26268.451} C_VEL
LIN {X 0,Y 282.726,Z 697.86,A -85,B 0,C 180,E1 26273.651,E2 26273.651} C_VEL
LIN {X 0,Y 281.218,Z 693.057,A -85,B 0,C 180,E1 26278.453,E2 26278.453} C_VEL
LIN {X 0,Y 280.654,Z 693.803,A -85,B 0,C 180,E1 26285.513,E2 26285.513} C_VEL
LIN {X 0,Y 282.341,Z 700.714,A -85,B 0,C 180,E1 26292.389,E2 26292.389} C_VEL
LIN {X 0,Y 286.739,Z 712.238,A -85,B 0,C 180,E1 26299.087,E2 26299.087} C_VEL
LIN {X 0,Y 292.218,Z 727.945,A -85,B 0,C 180,E1 26305.007,E2 26305.007} C_VEL
LIN {X 0,Y 296.755,Z 746.596,A -85,B 0,C 180,E1 26310.267,E2 26310.267} C_VEL
LIN {X 0,Y 298.368,Z 761.437,A -85,B 0,C 180,E1 26313.718,E2 26313.718} C_VEL
LIN {X 0,Y 296.317,Z 767.382,A -85,B 0,C 180,E1 26314.267,E2 26314.267} C_VEL
LIN {X 0,Y 287.901,Z 780.624,A -85,B 0,C 180,E1 26314.427,E2 26314.427} C_VEL
LIN {X 0,Y 287.271,Z 781.946,A -85,B 0,C 180,E1 26314.547,E2 26314.547} C_VEL
LIN {X 0,Y 271.697,Z 814.205,A -85,B 0,C 180,E1 26318.656,E2 26318.656} C_VEL
LIN {X 0,Y 254.924,Z 842.487,A -85,B 0,C 180,E1 26324.005,E2 26324.005} C_VEL
LIN {X 0,Y 238.642,Z 865.836,A -85,B 0,C 180,E1 26330.572,E2 26330.572} C_VEL
LIN {X 0,Y 224.482,Z 884.067,A -85,B 0,C 180,E1 26338.447,E2 26338.447} C_VEL
LIN {X 0,Y 213.577,Z 897.595,A -85,B 0,C 180,E1 26347.76,E2 26347.76} C_VEL
LIN {X 0,Y 207.35,Z 905.531,A -85,B 0,C 180,E1 26357.325,E2 26357.325} C_VEL
LIN {X 0,Y 205.172,Z 908.628,A -85,B 0,C 180,E1 26365.753,E2 26365.753} C_VEL
LIN {X 0,Y 205.272,Z 908.591,A -85,B 0,C 180,E1 26374.221,E2 26374.221} C_VEL
LIN {X 0,Y 208.406,Z 904.096,A -85,B 0,C 180,E1 26384.73,E2 26384.73} C_VEL
LIN {X 0,Y 216.255,Z 894.273,A -85,B 0,C 180,E1 26394.847,E2 26394.847} C_VEL
LIN {X 0,Y 229.025,Z 878.187,A -85,B 0,C 180,E1 26404.362,E2 26404.362} C_VEL
LIN {X 0,Y 244.537,Z 857.417,A -85,B 0,C 180,E1 26411.986,E2 26411.986} C_VEL
LIN {X 0,Y 261.917,Z 830.991,A -85,B 0,C 180,E1 26418.322,E2 26418.322} C_VEL
LIN {X 0,Y 267.56,Z 821.396,A -85,B 0,C 180,E1 26420.048,E2 26420.048} C_VEL
LIN {X 0,Y 267.947,Z 819.664,A -85,B 0,C 180,E1 26420.535,E2 26420.535} C_VEL
LIN {X 0,Y 239.009,Z 833.339,A -85,B 0,C 180,E1 26426.384,E2 26426.384} C_VEL
LIN {X 0,Y 212.482,Z 844.844,A -85,B 0,C 180,E1 26435.804,E2 26435.804} C_VEL
LIN {X 0,Y 211.418,Z 845.937,A -85,B 0,C 180,E1 26436.796,E2 26436.796} C_VEL
LIN {X 0,Y 206.51,Z 873.906,A -85,B 0,C 180,E1 26445.128,E2 26445.128} C_VEL
LIN {X 0,Y 204.558,Z 895.702,A -85,B 0,C 180,E1 26454.161,E2 26454.161} C_VEL
LIN {X 0,Y 205.478,Z 911.244,A -85,B 0,C 180,E1 26463.175,E2 26463.175} C_VEL
LIN {X 0,Y 210.573,Z 922.201,A -85,B 0,C 180,E1 26472.469,E2 26472.469} C_VEL
LIN {X 0,Y 219.004,Z 927.938,A -85,B 0,C 180,E1 26480.239,E2 26480.239} C_VEL
LIN {X 0,Y 238.793,Z 930.516,A -85,B 0,C 180,E1 26490.504,E2 26490.504} C_VEL
LIN {X 0,Y 257.65,Z 928.743,A -85,B 0,C 180,E1 26496.493,E2 26496.493} C_VEL
LIN {X 0,Y 251.724,Z 931.646,A -85,B 0,C 180,E1 26498.524,E2 26498.524} C_VEL
LIN {X 0,Y 220.234,Z 947.382,A -85,B 0,C 180,E1 26511.756,E2 26511.756} C_VEL
LIN {X 0,Y 205.017,Z 957.309,A -85,B 0,C 180,E1 26528.326,E2 26528.326} C_VEL
LIN {X 0,Y 203.54,Z 959.288,A -85,B 0,C 180,E1 26541.45,E2 26541.45} C_VEL
LIN {X 0,Y 204.619,Z 960.684,A -85,B 0,C 180,E1 26550.012,E2 26550.012} C_VEL
LIN {X 0,Y 203.651,Z 958.781,A -85,B 0,C 180,E1 26558.569,E2 26558.569} C_VEL
LIN {X 0,Y 204.015,Z 953.354,A -85,B 0,C 180,E1 26567.294,E2 26567.294} C_VEL
LIN {X 0,Y 208.578,Z 941.575,A -85,B 0,C 180,E1 26578.078,E2 26578.078} C_VEL
LIN {X 0,Y 219.331,Z 923.211,A -85,B 0,C 180,E1 26588.458,E2 26588.458} C_VEL
LIN {X 0,Y 233.831,Z 900.079,A -85,B 0,C 180,E1 26596.82,E2 26596.82} C_VEL
LIN {X 0,Y 250.195,Z 872.321,A -85,B 0,C 180,E1 26603.379,E2 26603.379} C_VEL
LIN {X 0,Y 266.018,Z 841.367,A -85,B 0,C 180,E1 26608.201,E2 26608.201} C_VEL
LIN {X 0,Y 280.061,Z 807.119,A -85,B 0,C 180,E1 26611.75,E2 26611.75} C_VEL
LIN {X 0,Y 290.135,Z 773.541,A -85,B 0,C 180,E1 26614.207,E2 26614.207} C_VEL
LIN {X 0,Y 289.117,Z 724.809,A -85,B 0,C 180,E1 26622.626,E2 26622.626} C_VEL
LIN {X 0,Y 283.45,Z 711.639,A -85,B 0,C 180,E1 26628.923,E2 26628.923} C_VEL
LIN {X 0,Y 280.219,Z 705.043,A -85,B 0,C 180,E1 26634.178,E2 26634.178} C_VEL
LIN {X 0,Y 278.877,Z 700.558,A -85,B 0,C 180,E1 26639.295,E2 26639.295} C_VEL
LIN {X 0,Y 278.395,Z 701.51,A -85,B 0,C 180,E1 26645.46,E2 26645.46} C_VEL
LIN {X 0,Y 279.769,Z 707.2,A -85,B 0,C 180,E1 26651.518,E2 26651.518} C_VEL
LIN {X 0,Y 283.765,Z 719.065,A -85,B 0,C 180,E1 26658.567,E2 26658.567} C_VEL
LIN {X 0,Y 288.932,Z 735.389,A -85,B 0,C 180,E1 26664.795,E2 26664.795} C_VEL
LIN {X 0,Y 292.458,Z 753.779,A -85,B 0,C 180,E1 26670.021,E2 26670.021} C_VEL
LIN {X 0,Y 293.076,Z 767.097,A -85,B 0,C 180,E1 26673.107,E2 26673.107} C_VEL
LIN {X 0,Y 287.271,Z 781.946,A -85,B 0,C 180,E1 26674.547,E2 26674.547} C_VEL
LIN {X 0,Y 278.75,Z 796.527,A -85,B 0,C 180,E1 26675.501,E2 26675.501} C_VEL
LIN {X 0,Y 269.546,Z 810.458,A -85,B 0,C 180,E1 26676.609,E2 26676.609} C_VEL
LIN {X 0,Y 252.127,Z 839.629,A -85,B 0,C 180,E1 26681.811,E2 26681.811} C_VEL
LIN {X 0,Y 234.882,Z 863.865,A -85,B 0,C 180,E1 26688.317,E2 26688.317} C_VEL
LIN {X 0,Y 219.276,Z 883.413,A -85,B 0,C 180,E1 26696.427,E2 26696.427} C_VEL
LIN {X 0,Y 207.642,Z 897.067,A -85,B 0,C 180,E1 26705.572,E2 26705.572} C_VEL
LIN {X 0,Y 200.728,Z 905.185,A -85,B 0,C 180,E1 26714.668,E2 26714.668} C_VEL
LIN {X 0,Y 197.351,Z 909.617,A -85,B 0,C 180,E1 26725.585,E2 26725.585} C_VEL
LIN {X 0,Y 197.449,Z 909.581,A -85,B 0,C 180,E1 26734.389,E2 26734.389} C_VEL
LIN {X 0,Y 200.804,Z 905.102,A -85,B 0,C 180,E1 26745.301,E2 26745.301} C_VEL
LIN {X 0,Y 209.128,Z 895.289,A -85,B 0,C 180,E1 26755.755,E2 26755.755} C_VEL
LIN {X 0,Y 221.332,Z 880.688,A -85,B 0,C 180,E1 26764.791,E2 26764.791} C_VEL
LIN {X 0,Y 237.642,Z 860.006,A -85,B 0,C 180,E1 26772.793,E2 26772.793} C_VEL
LIN {X 0,Y 255.41,Z 834.25,A -85,B 0,C 180,E1 26779.204,E2 26779.204} C_VEL
LIN {X 0,Y 258.448,Z 828.501,A -85,B 0,C 180,E1 26780.489,E2 26780.489} C_VEL
LIN {X 0,Y 226.619,Z 842.361,A -85,B 0,C 180,E1 26787.677,E2 26787.677} C_VEL
LIN {X 0,Y 205.365,Z 851.139,A -85,B 0,C 180,E1 26796.07,E2 26796.07} C_VEL
LIN {X 0,Y 202.198,Z 853.018,A -85,B 0,C 180,E1 26798.318,E2 26798.318} C_VEL
LIN {X 0,Y 197.86,Z 880.016,A -85,B 0,C 180,E1 26807.29,E2 26807.29} C_VEL
LIN {X 0,Y 196.682,Z 900.369,A -85,B 0,C 180,E1 26816.694,E2 26816.694} C_VEL
LIN {X 0,Y 198.752,Z 915.489,A -85,B 0,C 180,E1 26826.57,E2 26826.57} C_VEL
LIN {X 0,Y 206.755,Z 926.131,A -85,B 0,C 180,E1 26837.048,E2 26837.048} C_VEL
LIN {X 0,Y 217.527,Z 930.736,A -85,B 0,C 180,E1 26844.704,E2 26844.704} C_VEL
LIN {X 0,Y 240.87,Z 932.009,A -85,B 0,C 180,E1 26854.479,E2 26854.479} C_VEL
LIN {X 0,Y 247.686,Z 931.486,A -85,B 0,C 180,E1 26856.46,E2 26856.46} C_VEL
LIN {X 0,Y 242.558,Z 933.86,A -85,B 0,C 180,E1 26858.275,E2 26858.275} C_VEL
LIN {X 0,Y 211.22,Z 948.048,A -85,B 0,C 180,E1 26872.094,E2 26872.094} C_VEL
LIN {X 0,Y 197.493,Z 955.955,A -85,B 0,C 180,E1 26887.456,E2 26887.456} C_VEL
LIN {X 0,Y 195.748,Z 957.75,A -85,B 0,C 180,E1 26901.106,E2 26901.106} C_VEL
LIN {X 0,Y 196.763,Z 959.694,A -85,B 0,C 180,E1 26910.012,E2 26910.012} C_VEL
LIN {X 0,Y 195.772,Z 957.771,A -85,B 0,C 180,E1 26918.917,E2 26918.917} C_VEL
LIN {X 0,Y 196.815,Z 950.358,A -85,B 0,C 180,E1 26930.283,E2 26930.283} C_VEL
LIN {X 0,Y 203.204,Z 937.2,A -85,B 0,C 180,E1 26941.478,E2 26941.478} C_VEL
LIN {X 0,Y 215.667,Z 917.821,A -85,B 0,C 180,E1 26951.693,E2 26951.693} C_VEL
LIN {X 0,Y 231.072,Z 894.405,A -85,B 0,C 180,E1 26959.599,E2 26959.599} C_VEL
LIN {X 0,Y 248.254,Z 865.857,A -85,B 0,C 180,E1 26965.888,E2 26965.888} C_VEL
LIN {X 0,Y 264.627,Z 833.888,A -85,B 0,C 180,E1 26970.503,E2 26970.503} C_VEL
LIN {X 0,Y 278.695,Z 798.989,A -85,B 0,C 180,E1 26973.804,E2 26973.804} C_VEL
LIN {X 0,Y 285.464,Z 775.766,A -85,B 0,C 180,E1 26975.522,E2 26975.522} C_VEL
LIN {X 0,Y 285.774,Z 732.224,A -85,B 0,C 180,E1 26983.043,E2 26983.043} C_VEL
LIN {X 0,Y 281.201,Z 719.803,A -85,B 0,C 180,E1 26988.735,E2 26988.735} C_VEL
LIN {X 0,Y 277.904,Z 712.576,A -85,B 0,C 180,E1 26994.326,E2 26994.326} C_VEL
LIN {X 0,Y 276.629,Z 708.112,A -85,B 0,C 180,E1 26999.289,E2 26999.289} C_VEL
LIN {X 0,Y 276.126,Z 708.997,A -85,B 0,C 180,E1 27005.209,E2 27005.209} C_VEL
LIN {X 0,Y 278.125,Z 717.5,A -85,B 0,C 180,E1 27013.364,E2 27013.364} C_VEL
LIN {X 0,Y 281.941,Z 729.392,A -85,B 0,C 180,E1 27019.618,E2 27019.618} C_VEL
LIN {X 0,Y 285.976,Z 745.641,A -85,B 0,C 180,E1 27025.471,E2 27025.471} C_VEL
LIN {X 0,Y 288.26,Z 765.04,A -85,B 0,C 180,E1 27030.819,E2 27030.819} C_VEL
LIN {X 0,Y 288.213,Z 769.962,A -85,B 0,C 180,E1 27031.976,E2 27031.976} C_VEL
LIN {X 0,Y 273.337,Z 803.163,A -85,B 0,C 180,E1 27035.599,E2 27035.599} C_VEL
LIN {X 0,Y 269.546,Z 810.458,A -85,B 0,C 180,E1 27036.609,E2 27036.609} C_VEL
LIN {X 0,Y 259.901,Z 823.776,A -85,B 0,C 180,E1 27037.949,E2 27037.949} C_VEL
LIN {X 0,Y 249.934,Z 836.324,A -85,B 0,C 180,E1 27039.528,E2 27039.528} C_VEL
LIN {X 0,Y 231.385,Z 862.042,A -85,B 0,C 180,E1 27046.062,E2 27046.062} C_VEL
LIN {X 0,Y 214.669,Z 882.182,A -85,B 0,C 180,E1 27054.101,E2 27054.101} C_VEL
LIN {X 0,Y 201.986,Z 896.47,A -85,B 0,C 180,E1 27063.237,E2 27063.237} C_VEL
LIN {X 0,Y 193.151,Z 906.189,A -85,B 0,C 180,E1 27074.051,E2 27074.051} C_VEL
LIN {X 0,Y 189.54,Z 910.606,A -85,B 0,C 180,E1 27085.402,E2 27085.402} C_VEL
LIN {X 0,Y 189.637,Z 910.569,A -85,B 0,C 180,E1 27094.57,E2 27094.57} C_VEL
LIN {X 0,Y 193.225,Z 906.102,A -85,B 0,C 180,E1 27105.917,E2 27105.917} C_VEL
LIN {X 0,Y 202.053,Z 896.31,A -85,B 0,C 180,E1 27116.727,E2 27116.727} C_VEL
LIN {X 0,Y 216.015,Z 880.505,A -85,B 0,C 180,E1 27126.601,E2 27126.601} C_VEL
LIN {X 0,Y 232.644,Z 860.151,A -85,B 0,C 180,E1 27134.388,E2 27134.388} C_VEL
LIN {X 0,Y 248.052,Z 838.766,A -85,B 0,C 180,E1 27139.838,E2 27139.838} C_VEL
LIN {X 0,Y 248.579,Z 836.819,A -85,B 0,C 180,E1 27140.551,E2 27140.551} C_VEL
LIN {X 0,Y 216.684,Z 849.816,A -85,B 0,C 180,E1 27148.382,E2 27148.382} C_VEL
LIN {X 0,Y 193.611,Z 859.094,A -85,B 0,C 180,E1 27159.259,E2 27159.259} C_VEL
LIN {X 0,Y 193.009,Z 860.126,A -85,B 0,C 180,E1 27160.119,E2 27160.119} C_VEL
LIN {X 0,Y 189.375,Z 885.681,A -85,B 0,C 180,E1 27169.637,E2 27169.637} C_VEL
LIN {X 0,Y 189.035,Z 905.694,A -85,B 0,C 180,E1 27180.006,E2 27180.006} C_VEL
LIN {X 0,Y 193.57,Z 920.628,A -85,B 0,C 180,E1 27191.288,E2 27191.288} C_VEL
LIN {X 0,Y 204.376,Z 929.599,A -85,B 0,C 180,E1 27201.759,E2 27201.759} C_VEL
LIN {X 0,Y 225.634,Z 933.896,A -85,B 0,C 180,E1 27212.493,E2 27212.493} C_VEL
LIN {X 0,Y 236.847,Z 933.851,A -85,B 0,C 180,E1 27216.2,E2 27216.2} C_VEL
LIN {X 0,Y 236.139,Z 934.565,A -85,B 0,C 180,E1 27217.177,E2 27217.177} C_VEL
LIN {X 0,Y 204.802,Z 947.287,A -85,B 0,C 180,E1 27230.682,E2 27230.682} C_VEL
LIN {X 0,Y 190.027,Z 954.598,A -85,B 0,C 180,E1 27246.518,E2 27246.518} C_VEL
LIN {X 0,Y 187.854,Z 956.747,A -85,B 0,C 180,E1 27260.73,E2 27260.73} C_VEL
LIN {X 0,Y 188.918,Z 958.705,A -85,B 0,C 180,E1 27270.013,E2 27270.013} C_VEL
LIN {X 0,Y 187.886,Z 956.759,A -85,B 0,C 180,E1 27279.295,E2 27279.295} C_VEL
LIN {X 0,Y 189.176,Z 949.298,A -85,B 0,C 180,E1 27291.14,E2 27291.14} C_VEL
LIN {X 0,Y 196.224,Z 936.096,A -85,B 0,C 180,E1 27302.734,E2 27302.734} C_VEL
LIN {X 0,Y 208.717,Z 917.775,A -85,B 0,C 180,E1 27312.734,E2 27312.734} C_VEL
LIN {X 0,Y 225.271,Z 893.913,A -85,B 0,C 180,E1 27321.013,E2 27321.013} C_VEL
LIN {X 0,Y 243.087,Z 865.714,A -85,B 0,C 180,E1 27327.315,E2 27327.315} C_VEL
LIN {X 0,Y 260.063,Z 833.933,A -85,B 0,C 180,E1 27331.927,E2 27331.927} C_VEL
LIN {X 0,Y 274.984,Z 798.32,A -85,B 0,C 180,E1 27335.291,E2 27335.291} C_VEL
LIN {X 0,Y 281.032,Z 779.185,A -85,B 0,C 180,E1 27336.667,E2 27336.667} C_VEL
LIN {X 0,Y 282.203,Z 737.914,A -85,B 0,C 180,E1 27343.94,E2 27343.94} C_VEL
LIN {X 0,Y 277.926,Z 726.028,A -85,B 0,C 180,E1 27349.718,E2 27349.718} C_VEL
LIN {X 0,Y 275.167,Z 719.421,A -85,B 0,C 180,E1 27355.111,E2 27355.111} C_VEL
LIN {X 0,Y 274.18,Z 715.52,A -85,B 0,C 180,E1 27359.996,E2 27359.996} C_VEL
LIN {X 0,Y 273.829,Z 716.525,A -85,B 0,C 180,E1 27365.02,E2 27365.02} C_VEL
LIN {X 0,Y 275.336,Z 724.351,A -85,B 0,C 180,E1 27372.71,E2 27372.71} C_VEL
LIN {X 0,Y 278.245,Z 734.221,A -85,B 0,C 180,E1 27378.239,E2 27378.239} C_VEL
LIN {X 0,Y 281.598,Z 749.535,A -85,B 0,C 180,E1 27384.137,E2 27384.137} C_VEL
LIN {X 0,Y 283.43,Z 767.997,A -85,B 0,C 180,E1 27389.549,E2 27389.549} C_VEL
LIN {X 0,Y 282.747,Z 774.556,A -85,B 0,C 180,E1 27390.956,E2 27390.956} C_VEL
LIN {X 0,Y 266.845,Z 807.973,A -85,B 0,C 180,E1 27394.745,E2 27394.745} C_VEL
LIN {X 0,Y 249.934,Z 836.324,A -85,B 0,C 180,E1 27399.528,E2 27399.528} C_VEL
LIN {X 0,Y 239.554,Z 848.14,A -85,B 0,C 180,E1 27401.359,E2 27401.359} C_VEL
LIN {X 0,Y 228.956,Z 859.144,A -85,B 0,C 180,E1 27403.462,E2 27403.462} C_VEL
LIN {X 0,Y 211.263,Z 880.033,A -85,B 0,C 180,E1 27411.247,E2 27411.247} C_VEL
LIN {X 0,Y 196.178,Z 896.171,A -85,B 0,C 180,E1 27421.123,E2 27421.123} C_VEL
LIN {X 0,Y 187.066,Z 905.675,A -85,B 0,C 180,E1 27431.082,E2 27431.082} C_VEL
LIN {X 0,Y 182.647,Z 910.44,A -85,B 0,C 180,E1 27440.436,E2 27440.436} C_VEL
LIN {X 0,Y 181.659,Z 911.987,A -85,B 0,C 180,E1 27449.987,E2 27449.987} C_VEL
LIN {X 0,Y 182.731,Z 910.389,A -85,B 0,C 180,E1 27459.533,E2 27459.533} C_VEL
LIN {X 0,Y 188.797,Z 903.874,A -85,B 0,C 180,E1 27471.157,E2 27471.157} C_VEL
LIN {X 0,Y 200.295,Z 891.785,A -85,B 0,C 180,E1 27481.96,E2 27481.96} C_VEL
LIN {X 0,Y 216.153,Z 874.386,A -85,B 0,C 180,E1 27491.07,E2 27491.07} C_VEL
LIN {X 0,Y 234.896,Z 851.284,A -85,B 0,C 180,E1 27498.564,E2 27498.564} C_VEL
LIN {X 0,Y 239.666,Z 844.307,A -85,B 0,C 180,E1 27500.395,E2 27500.395} C_VEL
LIN {X 0,Y 206.764,Z 856.875,A -85,B 0,C 180,E1 27509.151,E2 27509.151} C_VEL
LIN {X 0,Y 184.05,Z 866.507,A -85,B 0,C 180,E1 27522.028,E2 27522.028} C_VEL
LIN {X 0,Y 181.068,Z 891.006,A -85,B 0,C 180,E1 27532.192,E2 27532.192} C_VEL
LIN {X 0,Y 181.488,Z 908.773,A -85,B 0,C 180,E1 27542.398,E2 27542.398} C_VEL
LIN {X 0,Y 187.552,Z 923.08,A -85,B 0,C 180,E1 27554.029,E2 27554.029} C_VEL
LIN {X 0,Y 200.168,Z 931.608,A -85,B 0,C 180,E1 27564.604,E2 27564.604} C_VEL
LIN {X 0,Y 219.129,Z 935.35,A -85,B 0,C 180,E1 27573.583,E2 27573.583} C_VEL
LIN {X 0,Y 227.107,Z 936.026,A -85,B 0,C 180,E1 27576.829,E2 27576.829} C_VEL
LIN {X 0,Y 194.981,Z 947.849,A -85,B 0,C 180,E1 27591.576,E2 27591.576} C_VEL
LIN {X 0,Y 182.37,Z 953.272,A -85,B 0,C 180,E1 27606.041,E2 27606.041} C_VEL
LIN {X 0,Y 180.099,Z 954.344,A -85,B 0,C 180,E1 27615.394,E2 27615.394} C_VEL
LIN {X 0,Y 180.364,Z 957.13,A -85,B 0,C 180,E1 27625.194,E2 27625.194} C_VEL
LIN {X 0,Y 181.065,Z 957.715,A -85,B 0,C 180,E1 27630.013,E2 27630.013} C_VEL
LIN {X 0,Y 179.988,Z 955.743,A -85,B 0,C 180,E1 27639.706,E2 27639.706} C_VEL
LIN {X 0,Y 181.444,Z 948.49,A -85,B 0,C 180,E1 27651.753,E2 27651.753} C_VEL
LIN {X 0,Y 189.304,Z 935.005,A -85,B 0,C 180,E1 27664.091,E2 27664.091} C_VEL
LIN {X 0,Y 202.489,Z 916.865,A -85,B 0,C 180,E1 27674.221,E2 27674.221} C_VEL
LIN {X 0,Y 219.229,Z 894.057,A -85,B 0,C 180,E1 27682.331,E2 27682.331} C_VEL
LIN {X 0,Y 237.97,Z 865.774,A -85,B 0,C 180,E1 27688.757,E2 27688.757} C_VEL
LIN {X 0,Y 255.545,Z 834.295,A -85,B 0,C 180,E1 27693.368,E2 27693.368} C_VEL
LIN {X 0,Y 270.793,Z 799.503,A -85,B 0,C 180,E1 27696.671,E2 27696.671} C_VEL
LIN {X 0,Y 276.624,Z 782.402,A -85,B 0,C 180,E1 27697.882,E2 27697.882} C_VEL
LIN {X 0,Y 278.638,Z 743.003,A -85,B 0,C 180,E1 27705.03,E2 27705.03} C_VEL
LIN {X 0,Y 274.599,Z 731.897,A -85,B 0,C 180,E1 27711.07,E2 27711.07} C_VEL
LIN {X 0,Y 272.493,Z 726.242,A -85,B 0,C 180,E1 27716.061,E2 27716.061} C_VEL
LIN {X 0,Y 271.909,Z 723.071,A -85,B 0,C 180,E1 27719.996,E2 27719.996} C_VEL
LIN {X 0,Y 271.391,Z 724.253,A -85,B 0,C 180,E1 27725.065,E2 27725.065} C_VEL
LIN {X 0,Y 272.762,Z 731.961,A -85,B 0,C 180,E1 27732.628,E2 27732.628} C_VEL
LIN {X 0,Y 275.777,Z 744.431,A -85,B 0,C 180,E1 27739.24,E2 27739.24} C_VEL
LIN {X 0,Y 278.098,Z 759.819,A -85,B 0,C 180,E1 27744.915,E2 27744.915} C_VEL
LIN {X 0,Y 278.542,Z 775.67,A -85,B 0,C 180,E1 27749.482,E2 27749.482} C_VEL
LIN {X 0,Y 262.466,Z 809.041,A -85,B 0,C 180,E1 27753.342,E2 27753.342} C_VEL
LIN {X 0,Y 244.367,Z 838.322,A -85,B 0,C 180,E1 27758.305,E2 27758.305} C_VEL
LIN {X 0,Y 228.956,Z 859.144,A -85,B 0,C 180,E1 27763.462,E2 27763.462} C_VEL
LIN {X 0,Y 218.206,Z 869.301,A -85,B 0,C 180,E1 27765.894,E2 27765.894} C_VEL
LIN {X 0,Y 207.586,Z 878.525,A -85,B 0,C 180,E1 27768.699,E2 27768.699} C_VEL
LIN {X 0,Y 190.718,Z 895.894,A -85,B 0,C 180,E1 27778.894,E2 27778.894} C_VEL
LIN {X 0,Y 179.637,Z 906.675,A -85,B 0,C 180,E1 27790.268,E2 27790.268} C_VEL
LIN {X 0,Y 174.909,Z 911.432,A -85,B 0,C 180,E1 27800.009,E2 27800.009} C_VEL
LIN {X 0,Y 173.834,Z 912.974,A -85,B 0,C 180,E1 27809.986,E2 27809.986} C_VEL
LIN {X 0,Y 174.991,Z 911.385,A -85,B 0,C 180,E1 27819.959,E2 27819.959} C_VEL
LIN {X 0,Y 181.478,Z 904.88,A -85,B 0,C 180,E1 27832.054,E2 27832.054} C_VEL
LIN {X 0,Y 193.65,Z 892.822,A -85,B 0,C 180,E1 27843.195,E2 27843.195} C_VEL
LIN {X 0,Y 210.286,Z 875.43,A -85,B 0,C 180,E1 27852.478,E2 27852.478} C_VEL
LIN {X 0,Y 229.041,Z 853.278,A -85,B 0,C 180,E1 27859.788,E2 27859.788} C_VEL
LIN {X 0,Y 229.954,Z 851.634,A -85,B 0,C 180,E1 27860.372,E2 27860.372} C_VEL
LIN {X 0,Y 196.849,Z 863.588,A -85,B 0,C 180,E1 27869.992,E2 27869.992} C_VEL
LIN {X 0,Y 175.073,Z 873.003,A -85,B 0,C 180,E1 27884.318,E2 27884.318} C_VEL
LIN {X 0,Y 173.006,Z 896.029,A -85,B 0,C 180,E1 27894.983,E2 27894.983} C_VEL
LIN {X 0,Y 174.688,Z 913.446,A -85,B 0,C 180,E1 27906.229,E2 27906.229} C_VEL
LIN {X 0,Y 181.975,Z 925.47,A -85,B 0,C 180,E1 27916.946,E2 27916.946} C_VEL
LIN {X 0,Y 196.435,Z 933.609,A -85,B 0,C 180,E1 27927.569,E2 27927.569} C_VEL
LIN {X 0,Y 216.677,Z 937.259,A -85,B 0,C 180,E1 27936.384,E2 27936.384} C_VEL
LIN {X 0,Y 202.806,Z 942.035,A -85,B 0,C 180,E1 27942.249,E2 27942.249} C_VEL
LIN {X 0,Y 178.468,Z 950.367,A -85,B 0,C 180,E1 27959.392,E2 27959.392} C_VEL
LIN {X 0,Y 172.392,Z 952.63,A -85,B 0,C 180,E1 27975.178,E2 27975.178} C_VEL
LIN {X 0,Y 172.481,Z 956.132,A -85,B 0,C 180,E1 27984.974,E2 27984.974} C_VEL
LIN {X 0,Y 173.215,Z 956.725,A -85,B 0,C 180,E1 27990.014,E2 27990.014} C_VEL
LIN {X 0,Y 172.108,Z 954.729,A -85,B 0,C 180,E1 28000.155,E2 28000.155} C_VEL
LIN {X 0,Y 173.815,Z 947.564,A -85,B 0,C 180,E1 28012.59,E2 28012.59} C_VEL
LIN {X 0,Y 182.494,Z 933.894,A -85,B 0,C 180,E1 28025.551,E2 28025.551} C_VEL
LIN {X 0,Y 197.192,Z 914.97,A -85,B 0,C 180,E1 28036.251,E2 28036.251} C_VEL
LIN {X 0,Y 215.869,Z 890.662,A -85,B 0,C 180,E1 28044.702,E2 28044.702} C_VEL
LIN {X 0,Y 235.483,Z 861.85,A -85,B 0,C 180,E1 28050.949,E2 28050.949} C_VEL
LIN {X 0,Y 253.686,Z 829.716,A -85,B 0,C 180,E1 28055.388,E2 28055.388} C_VEL
LIN {X 0,Y 269.401,Z 793.657,A -85,B 0,C 180,E1 28058.61,E2 28058.61} C_VEL
LIN {X 0,Y 272.416,Z 784.472,A -85,B 0,C 180,E1 28059.337,E2 28059.337} C_VEL
LIN {X 0,Y 275.015,Z 748.56,A -85,B 0,C 180,E1 28066.051,E2 28066.051} C_VEL
LIN {X 0,Y 271.508,Z 738.358,A -85,B 0,C 180,E1 28071.978,E2 28071.978} C_VEL
LIN {X 0,Y 269.564,Z 731.569,A -85,B 0,C 180,E1 28078.386,E2 28078.386} C_VEL
LIN {X 0,Y 269.089,Z 730.782,A -85,B 0,C 180,E1 28083.223,E2 28083.223} C_VEL
LIN {X 0,Y 269.804,Z 737.962,A -85,B 0,C 180,E1 28091.329,E2 28091.329} C_VEL
LIN {X 0,Y 271.696,Z 747.402,A -85,B 0,C 180,E1 28097.018,E2 28097.018} C_VEL
LIN {X 0,Y 273.524,Z 761.45,A -85,B 0,C 180,E1 28102.806,E2 28102.806} C_VEL
LIN {X 0,Y 273.838,Z 778.312,A -85,B 0,C 180,E1 28108.074,E2 28108.074} C_VEL
LIN {X 0,Y 270.988,Z 785.669,A -85,B 0,C 180,E1 28109.036,E2 28109.036} C_VEL
LIN {X 0,Y 254.207,Z 817.037,A -85,B 0,C 180,E1 28112.884,E2 28112.884} C_VEL
LIN {X 0,Y 235.676,Z 844.836,A -85,B 0,C 180,E1 28118.011,E2 28118.011} C_VEL
LIN {X 0,Y 216.391,Z 868.694,A -85,B 0,C 180,E1 28124.763,E2 28124.763} C_VEL
LIN {X 0,Y 207.586,Z 878.525,A -85,B 0,C 180,E1 28128.699,E2 28128.699} C_VEL
LIN {X 0,Y 197.07,Z 886.854,A -85,B 0,C 180,E1 28131.907,E2 28131.907} C_VEL
LIN {X 0,Y 186.871,Z 894.175,A -85,B 0,C 180,E1 28135.555,E2 28135.555} C_VEL
LIN {X 0,Y 174.142,Z 906.019,A -85,B 0,C 180,E1 28146.954,E2 28146.954} C_VEL
LIN {X 0,Y 167.199,Z 912.424,A -85,B 0,C 180,E1 28159.543,E2 28159.543} C_VEL
LIN {X 0,Y 166.003,Z 913.961,A -85,B 0,C 180,E1 28169.986,E2 28169.986} C_VEL
LIN {X 0,Y 167.266,Z 912.38,A -85,B 0,C 180,E1 28180.424,E2 28180.424} C_VEL
LIN {X 0,Y 174.205,Z 905.887,A -85,B 0,C 180,E1 28193.027,E2 28193.027} C_VEL
LIN {X 0,Y 187.105,Z 893.844,A -85,B 0,C 180,E1 28204.517,E2 28204.517} C_VEL
LIN {X 0,Y 204.555,Z 876.489,A -85,B 0,C 180,E1 28213.966,E2 28213.966} C_VEL
LIN {X 0,Y 220.226,Z 858.502,A -85,B 0,C 180,E1 28220.362,E2 28220.362} C_VEL
LIN {X 0,Y 187.078,Z 869.87,A -85,B 0,C 180,E1 28230.938,E2 28230.938} C_VEL
LIN {X 0,Y 166.32,Z 879.112,A -85,B 0,C 180,E1 28246.845,E2 28246.845} C_VEL
LIN {X 0,Y 165.205,Z 900.615,A -85,B 0,C 180,E1 28258.036,E2 28258.036} C_VEL
LIN {X 0,Y 168.786,Z 917.734,A -85,B 0,C 180,E1 28270.347,E2 28270.347} C_VEL
LIN {X 0,Y 179.627,Z 929.659,A -85,B 0,C 180,E1 28282.31,E2 28282.31} C_VEL
LIN {X 0,Y 199.796,Z 937.042,A -85,B 0,C 180,E1 28293.488,E2 28293.488} C_VEL
LIN {X 0,Y 207.277,Z 938.295,A -85,B 0,C 180,E1 28296.495,E2 28296.495} C_VEL
LIN {X 0,Y 176.347,Z 947.345,A -85,B 0,C 180,E1 28313.043,E2 28313.043} C_VEL
LIN {X 0,Y 165.156,Z 950.71,A -85,B 0,C 180,E1 28331.286,E2 28331.286} C_VEL
LIN {X 0,Y 164.576,Z 955.129,A -85,B 0,C 180,E1 28344.732,E2 28344.732} C_VEL
LIN {X 0,Y 165.342,Z 955.733,A -85,B 0,C 180,E1 28350.014,E2 28350.014} C_VEL
LIN {X 0,Y 164.22,Z 953.712,A -85,B 0,C 180,E1 28360.649,E2 28360.649} C_VEL
LIN {X 0,Y 166.664,Z 945.797,A -85,B 0,C 180,E1 28374.624,E2 28374.624} C_VEL
LIN {X 0,Y 175.802,Z 932.781,A -85,B 0,C 180,E1 28387.125,E2 28387.125} C_VEL
LIN {X 0,Y 191.499,Z 913.831,A -85,B 0,C 180,E1 28398.061,E2 28398.061} C_VEL
LIN {X 0,Y 211.172,Z 889.458,A -85,B 0,C 180,E1 28406.545,E2 28406.545} C_VEL
LIN {X 0,Y 230.913,Z 861.728,A -85,B 0,C 180,E1 28412.552,E2 28412.552} C_VEL
LIN {X 0,Y 249.498,Z 830.262,A -85,B 0,C 180,E1 28416.906,E2 28416.906} C_VEL
LIN {X 0,Y 265.984,Z 793.964,A -85,B 0,C 180,E1 28420.136,E2 28420.136} C_VEL
LIN {X 0,Y 268.295,Z 786.404,A -85,B 0,C 180,E1 28420.877,E2 28420.877} C_VEL
LIN {X 0,Y 271.629,Z 755.31,A -85,B 0,C 180,E1 28426.676,E2 28426.676} C_VEL
LIN {X 0,Y 268.909,Z 746.106,A -85,B 0,C 180,E1 28431.9,E2 28431.9} C_VEL
LIN {X 0,Y 266.973,Z 738.178,A -85,B 0,C 180,E1 28439.996,E2 28439.996} C_VEL
LIN {X 0,Y 266.4,Z 739.361,A -85,B 0,C 180,E1 28444.889,E2 28444.889} C_VEL
LIN {X 0,Y 267.338,Z 746.841,A -85,B 0,C 180,E1 28452.264,E2 28452.264} C_VEL
LIN {X 0,Y 268.787,Z 758.331,A -85,B 0,C 180,E1 28458.479,E2 28458.479} C_VEL
LIN {X 0,Y 269.574,Z 774.105,A -85,B 0,C 180,E1 28464.471,E2 28464.471} C_VEL
LIN {X 0,Y 268.915,Z 783.326,A -85,B 0,C 180,E1 28467.227,E2 28467.227} C_VEL
LIN {X 0,Y 251.908,Z 815.12,A -85,B 0,C 180,E1 28470.928,E2 28470.928} C_VEL
LIN {X 0,Y 233.409,Z 842.528,A -85,B 0,C 180,E1 28475.735,E2 28475.735} C_VEL
LIN {X 0,Y 213.449,Z 867.02,A -85,B 0,C 180,E1 28482.282,E2 28482.282} C_VEL
LIN {X 0,Y 193.819,Z 887.532,A -85,B 0,C 180,E1 28491.272,E2 28491.272} C_VEL
LIN {X 0,Y 186.871,Z 894.175,A -85,B 0,C 180,E1 28495.555,E2 28495.555} C_VEL
LIN {X 0,Y 177.189,Z 900.576,A -85,B 0,C 180,E1 28499.711,E2 28499.711} C_VEL
LIN {X 0,Y 168.214,Z 905.87,A -85,B 0,C 180,E1 28504.396,E2 28504.396} C_VEL
LIN {X 0,Y 161.68,Z 911.511,A -85,B 0,C 180,E1 28513.656,E2 28513.656} C_VEL
LIN {X 0,Y 158.314,Z 914.56,A -85,B 0,C 180,E1 28524.493,E2 28524.493} C_VEL
LIN {X 0,Y 158.416,Z 914.524,A -85,B 0,C 180,E1 28535.473,E2 28535.473} C_VEL
LIN {X 0,Y 163.215,Z 910.113,A -85,B 0,C 180,E1 28548.945,E2 28548.945} C_VEL
LIN {X 0,Y 174.5,Z 900.385,A -85,B 0,C 180,E1 28561.382,E2 28561.382} C_VEL
LIN {X 0,Y 191.668,Z 884.718,A -85,B 0,C 180,E1 28572.201,E2 28572.201} C_VEL
LIN {X 0,Y 209.572,Z 866.352,A -85,B 0,C 180,E1 28579.746,E2 28579.746} C_VEL
LIN {X 0,Y 209.935,Z 865.184,A -85,B 0,C 180,E1 28580.461,E2 28580.461} C_VEL
LIN {X 0,Y 181.429,Z 874.462,A -85,B 0,C 180,E1 28589.942,E2 28589.942} C_VEL
LIN {X 0,Y 157.915,Z 884.14,A -85,B 0,C 180,E1 28608.946,E2 28608.946} C_VEL
LIN {X 0,Y 157.654,Z 904.995,A -85,B 0,C 180,E1 28621.383,E2 28621.383} C_VEL
LIN {X 0,Y 163.684,Z 921.701,A -85,B 0,C 180,E1 28634.751,E2 28634.751} C_VEL
LIN {X 0,Y 178.971,Z 933.425,A -85,B 0,C 180,E1 28647.752,E2 28647.752} C_VEL
LIN {X 0,Y 196.649,Z 938.663,A -85,B 0,C 180,E1 28656.056,E2 28656.056} C_VEL
LIN {X 0,Y 193.022,Z 940.037,A -85,B 0,C 180,E1 28658.3,E2 28658.3} C_VEL
LIN {X 0,Y 164.7,Z 947.192,A -85,B 0,C 180,E1 28676.514,E2 28676.514} C_VEL
LIN {X 0,Y 157.645,Z 948.829,A -85,B 0,C 180,E1 28690.358,E2 28690.358} C_VEL
LIN {X 0,Y 156.687,Z 954.126,A -85,B 0,C 180,E1 28704.466,E2 28704.466} C_VEL
LIN {X 0,Y 157.486,Z 954.742,A -85,B 0,C 180,E1 28710.015,E2 28710.015} C_VEL
LIN {X 0,Y 156.342,Z 952.694,A -85,B 0,C 180,E1 28721.192,E2 28721.192} C_VEL
LIN {X 0,Y 159.217,Z 944.729,A -85,B 0,C 180,E1 28735.859,E2 28735.859} C_VEL
LIN {X 0,Y 169.257,Z 931.685,A -85,B 0,C 180,E1 28748.821,E2 28748.821} C_VEL
LIN {X 0,Y 186.011,Z 912.686,A -85,B 0,C 180,E1 28759.969,E2 28759.969} C_VEL
LIN {X 0,Y 206.722,Z 888.285,A -85,B 0,C 180,E1 28768.46,E2 28768.46} C_VEL
LIN {X 0,Y 228.028,Z 859.299,A -85,B 0,C 180,E1 28774.609,E2 28774.609} C_VEL
LIN {X 0,Y 246.951,Z 828.045,A -85,B 0,C 180,E1 28778.752,E2 28778.752} C_VEL
LIN {X 0,Y 263.138,Z 793.193,A -85,B 0,C 180,E1 28781.767,E2 28781.767} C_VEL
LIN {X 0,Y 265.025,Z 783.503,A -85,B 0,C 180,E1 28783.389,E2 28783.389} C_VEL
LIN {X 0,Y 268.102,Z 760.725,A -85,B 0,C 180,E1 28787.714,E2 28787.714} C_VEL
LIN {X 0,Y 265.571,Z 751.634,A -85,B 0,C 180,E1 28793.445,E2 28793.445} C_VEL
LIN {X 0,Y 264.316,Z 745.691,A -85,B 0,C 180,E1 28799.996,E2 28799.996} C_VEL
LIN {X 0,Y 264.011,Z 745.889,A -85,B 0,C 180,E1 28803.285,E2 28803.285} C_VEL
LIN {X 0,Y 264.082,Z 752.53,A -85,B 0,C 180,E1 28810.824,E2 28810.824} C_VEL
LIN {X 0,Y 264.943,Z 761.984,A -85,B 0,C 180,E1 28816.608,E2 28816.608} C_VEL
LIN {X 0,Y 265.22,Z 776.22,A -85,B 0,C 180,E1 28822.54,E2 28822.54} C_VEL
LIN {X 0,Y 264.414,Z 786.423,A -85,B 0,C 180,E1 28825.906,E2 28825.906} C_VEL
LIN {X 0,Y 246.335,Z 818.838,A -85,B 0,C 180,E1 28829.76,E2 28829.76} C_VEL
LIN {X 0,Y 225.592,Z 847.961,A -85,B 0,C 180,E1 28835.097,E2 28835.097} C_VEL
LIN {X 0,Y 204.363,Z 872.124,A -85,B 0,C 180,E1 28842.129,E2 28842.129} C_VEL
LIN {X 0,Y 184.505,Z 891.488,A -85,B 0,C 180,E1 28851.571,E2 28851.571} C_VEL
LIN {X 0,Y 169.176,Z 905.074,A -85,B 0,C 180,E1 28863.38,E2 28863.38} C_VEL
LIN {X 0,Y 168.214,Z 905.87,A -85,B 0,C 180,E1 28864.396,E2 28864.396} C_VEL
LIN {X 0,Y 160.062,Z 910.225,A -85,B 0,C 180,E1 28869.605,E2 28869.605} C_VEL
LIN {X 0,Y 152.893,Z 913.373,A -85,B 0,C 180,E1 28875.371,E2 28875.371} C_VEL
LIN {X 0,Y 150.342,Z 915.935,A -85,B 0,C 180,E1 28889.984,E2 28889.984} C_VEL
LIN {X 0,Y 151.84,Z 914.368,A -85,B 0,C 180,E1 28901.496,E2 28901.496} C_VEL
LIN {X 0,Y 159.348,Z 908.319,A -85,B 0,C 180,E1 28914.663,E2 28914.663} C_VEL
LIN {X 0,Y 174.357,Z 895.916,A -85,B 0,C 180,E1 28927.451,E2 28927.451} C_VEL
LIN {X 0,Y 193.522,Z 878.596,A -85,B 0,C 180,E1 28937.207,E2 28937.207} C_VEL
LIN {X 0,Y 199.21,Z 872.932,A -85,B 0,C 180,E1 28939.499,E2 28939.499} C_VEL
LIN {X 0,Y 200.037,Z 871.357,A -85,B 0,C 180,E1 28940.467,E2 28940.467} C_VEL
LIN {X 0,Y 171.517,Z 880.188,A -85,B 0,C 180,E1 28950.944,E2 28950.944} C_VEL
LIN {X 0,Y 149.557,Z 890.085,A -85,B 0,C 180,E1 28972.733,E2 28972.733} C_VEL
LIN {X 0,Y 150.339,Z 908.053,A -85,B 0,C 180,E1 28984.341,E2 28984.341} C_VEL
LIN {X 0,Y 158.266,Z 924.136,A -85,B 0,C 180,E1 28998.132,E2 28998.132} C_VEL
LIN {X 0,Y 175.84,Z 935.448,A -85,B 0,C 180,E1 29011.132,E2 29011.132} C_VEL
LIN {X 0,Y 187.355,Z 938.925,A -85,B 0,C 180,E1 29016.312,E2 29016.312} C_VEL
LIN {X 0,Y 158.009,Z 945.476,A -85,B 0,C 180,E1 29034.893,E2 29034.893} C_VEL
LIN {X 0,Y 150.564,Z 946.951,A -85,B 0,C 180,E1 29047.846,E2 29047.846} C_VEL
LIN {X 0,Y 148.512,Z 951.673,A -85,B 0,C 180,E1 29058.242,E2 29058.242} C_VEL
LIN {X 0,Y 149.633,Z 953.752,A -85,B 0,C 180,E1 29070.016,E2 29070.016} C_VEL
LIN {X 0,Y 148.475,Z 951.676,A -85,B 0,C 180,E1 29081.793,E2 29081.793} C_VEL
LIN {X 0,Y 151.118,Z 944.827,A -85,B 0,C 180,E1 29095.534,E2 29095.534} C_VEL
LIN {X 0,Y 161.403,Z 932.236,A -85,B 0,C 180,E1 29109.341,E2 29109.341} C_VEL
LIN {X 0,Y 178.266,Z 914.269,A -85,B 0,C 180,E1 29120.731,E2 29120.731} C_VEL
LIN {X 0,Y 199.672,Z 890.5,A -85,B 0,C 180,E1 29129.538,E2 29129.538} C_VEL
LIN {X 0,Y 221.534,Z 862.478,A -85,B 0,C 180,E1 29135.772,E2 29135.772} C_VEL
LIN {X 0,Y 241.731,Z 830.895,A -85,B 0,C 180,E1 29140.118,E2 29140.118} C_VEL
LIN {X 0,Y 259.347,Z 795.159,A -85,B 0,C 180,E1 29143.247,E2 29143.247} C_VEL
LIN {X 0,Y 264.532,Z 767.694,A -85,B 0,C 180,E1 29148.432,E2 29148.432} C_VEL
LIN {X 0,Y 263.097,Z 760.45,A -85,B 0,C 180,E1 29152.552,E2 29152.552} C_VEL
LIN {X 0,Y 261.745,Z 753.24,A -85,B 0,C 180,E1 29159.996,E2 29159.996} C_VEL
LIN {X 0,Y 261.293,Z 753.42,A -85,B 0,C 180,E1 29163.319,E2 29163.319} C_VEL
LIN {X 0,Y 261.038,Z 760.208,A -85,B 0,C 180,E1 29170.952,E2 29170.952} C_VEL
LIN {X 0,Y 261.231,Z 771.281,A -85,B 0,C 180,E1 29177.405,E2 29177.405} C_VEL
LIN {X 0,Y 260.399,Z 786.402,A -85,B 0,C 180,E1 29183.432,E2 29183.432} C_VEL
LIN {X 0,Y 259.89,Z 789.81,A -85,B 0,C 180,E1 29184.557,E2 29184.557} C_VEL
LIN {X 0,Y 241.283,Z 821.802,A -85,B 0,C 180,E1 29188.437,E2 29188.437} C_VEL
LIN {X 0,Y 220.431,Z 849.944,A -85,B 0,C 180,E1 29193.643,E2 29193.643} C_VEL
LIN {X 0,Y 198.016,Z 874.384,A -85,B 0,C 180,E1 29200.901,E2 29200.901} C_VEL
LIN {X 0,Y 178.245,Z 892.663,A -85,B 0,C 180,E1 29210.101,E2 29210.101} C_VEL
LIN {X 0,Y 162.175,Z 906.087,A -85,B 0,C 180,E1 29222.134,E2 29222.134} C_VEL
LIN {X 0,Y 152.893,Z 913.373,A -85,B 0,C 180,E1 29235.371,E2 29235.371} C_VEL
LIN {X 0,Y 150.461,Z 914.613,A -85,B 0,C 180,E1 29238.516,E2 29238.516} C_VEL
LIN {X 0,Y 142.496,Z 916.822,A -85,B 0,C 180,E1 29247.45,E2 29247.45} C_VEL
LIN {X 0,Y 142.415,Z 916.818,A -85,B 0,C 180,E1 29248.333,E2 29248.333} C_VEL
LIN {X 0,Y 144.153,Z 915.364,A -85,B 0,C 180,E1 29262.118,E2 29262.118} C_VEL
LIN {X 0,Y 152.82,Z 908.866,A -85,B 0,C 180,E1 29276.556,E2 29276.556} C_VEL
LIN {X 0,Y 168.162,Z 896.955,A -85,B 0,C 180,E1 29289.085,E2 29289.085} C_VEL
LIN {X 0,Y 189.081,Z 878.878,A -85,B 0,C 180,E1 29299.296,E2 29299.296} C_VEL
LIN {X 0,Y 190.229,Z 877.168,A -85,B 0,C 180,E1 29300.433,E2 29300.433} C_VEL
LIN {X 0,Y 157.851,Z 886.925,A -85,B 0,C 180,E1 29314.422,E2 29314.422} C_VEL
LIN {X 0,Y 141.566,Z 896.24,A -85,B 0,C 180,E1 29336.941,E2 29336.941} C_VEL
LIN {X 0,Y 144.769,Z 914.588,A -85,B 0,C 180,E1 29350.559,E2 29350.559} C_VEL
LIN {X 0,Y 156.371,Z 928.881,A -85,B 0,C 180,E1 29364.321,E2 29364.321} C_VEL
LIN {X 0,Y 173.439,Z 937.43,A -85,B 0,C 180,E1 29374.6,E2 29374.6} C_VEL
LIN {X 0,Y 177.133,Z 938.878,A -85,B 0,C 180,E1 29376.781,E2 29376.781} C_VEL
LIN {X 0,Y 151.508,Z 943.538,A -85,B 0,C 180,E1 29393.146,E2 29393.146} C_VEL
LIN {X 0,Y 143.72,Z 945.034,A -85,B 0,C 180,E1 29405.076,E2 29405.076} C_VEL
LIN {X 0,Y 140.678,Z 950.656,A -85,B 0,C 180,E1 29417.578,E2 29417.578} C_VEL
LIN {X 0,Y 141.768,Z 952.761,A -85,B 0,C 180,E1 29430.017,E2 29430.017} C_VEL
LIN {X 0,Y 140.607,Z 950.655,A -85,B 0,C 180,E1 29442.464,E2 29442.464} C_VEL
LIN {X 0,Y 143.723,Z 943.77,A -85,B 0,C 180,E1 29456.951,E2 29456.951} C_VEL
LIN {X 0,Y 155.063,Z 931.141,A -85,B 0,C 180,E1 29471.288,E2 29471.288} C_VEL
LIN {X 0,Y 173.292,Z 912.955,A -85,B 0,C 180,E1 29482.949,E2 29482.949} C_VEL
LIN {X 0,Y 195.694,Z 889.214,A -85,B 0,C 180,E1 29491.667,E2 29491.667} C_VEL
LIN {X 0,Y 218.276,Z 861.254,A -85,B 0,C 180,E1 29497.749,E2 29497.749} C_VEL
LIN {X 0,Y 239.078,Z 829.698,A -85,B 0,C 180,E1 29501.958,E2 29501.958} C_VEL
LIN {X 0,Y 256.338,Z 795.26,A -85,B 0,C 180,E1 29505.049,E2 29505.049} C_VEL
LIN {X 0,Y 260.994,Z 773.513,A -85,B 0,C 180,E1 29509.401,E2 29509.401} C_VEL
LIN {X 0,Y 259.879,Z 767.015,A -85,B 0,C 180,E1 29513.301,E2 29513.301} C_VEL
LIN {X 0,Y 258.923,Z 760.691,A -85,B 0,C 180,E1 29519.996,E2 29519.996} C_VEL
LIN {X 0,Y 258.051,Z 762.049,A -85,B 0,C 180,E1 29525.046,E2 29525.046} C_VEL
LIN {X 0,Y 257.652,Z 768.938,A -85,B 0,C 180,E1 29531.871,E2 29531.871} C_VEL
LIN {X 0,Y 257.102,Z 780.461,A -85,B 0,C 180,E1 29538.18,E2 29538.18} C_VEL
LIN {X 0,Y 255.334,Z 793.763,A -85,B 0,C 180,E1 29543.288,E2 29543.288} C_VEL
LIN {X 0,Y 236.185,Z 825.01,A -85,B 0,C 180,E1 29547.089,E2 29547.089} C_VEL
LIN {X 0,Y 214.993,Z 852.357,A -85,B 0,C 180,E1 29552.23,E2 29552.23} C_VEL
LIN {X 0,Y 193.304,Z 875.086,A -85,B 0,C 180,E1 29558.996,E2 29558.996} C_VEL
LIN {X 0,Y 172.286,Z 893.704,A -85,B 0,C 180,E1 29568.423,E2 29568.423} C_VEL
LIN {X 0,Y 155.252,Z 907.104,A -85,B 0,C 180,E1 29580.774,E2 29580.774} C_VEL
LIN {X 0,Y 145.197,Z 914.444,A -85,B 0,C 180,E1 29594.826,E2 29594.826} C_VEL
LIN {X 0,Y 142.415,Z 916.818,A -85,B 0,C 180,E1 29608.333,E2 29608.333} C_VEL
LIN {X 0,Y 140.107,Z 917.11,A -85,B 0,C 180,E1 29613.561,E2 29613.561} C_VEL
LIN {X 0,Y 136.202,Z 916.601,A -85,B 0,C 180,E1 29621.675,E2 29621.675} C_VEL
LIN {X 0,Y 136.419,Z 916.397,A -85,B 0,C 180,E1 29622.598,E2 29622.598} C_VEL
LIN {X 0,Y 144.921,Z 910.523,A -85,B 0,C 180,E1 29636.954,E2 29636.954} C_VEL
LIN {X 0,Y 160.188,Z 899.428,A -85,B 0,C 180,E1 29649.659,E2 29649.659} C_VEL
LIN {X 0,Y 179.596,Z 883.883,A -85,B 0,C 180,E1 29659.383,E2 29659.383} C_VEL
LIN {X 0,Y 180.786,Z 882.521,A -85,B 0,C 180,E1 29660.269,E2 29660.269} C_VEL
LIN {X 0,Y 144.967,Z 893.275,A -85,B 0,C 180,E1 29678.555,E2 29678.555} C_VEL
LIN {X 0,Y 134.117,Z 901.943,A -85,B 0,C 180,E1 29701.626,E2 29701.626} C_VEL
LIN {X 0,Y 140.945,Z 920.476,A -85,B 0,C 180,E1 29717.2,E2 29717.2} C_VEL
LIN {X 0,Y 158.41,Z 934.194,A -85,B 0,C 180,E1 29731.742,E2 29731.742} C_VEL
LIN {X 0,Y 166.968,Z 937.768,A -85,B 0,C 180,E1 29736.147,E2 29736.147} C_VEL
LIN {X 0,Y 159.662,Z 939.447,A -85,B 0,C 180,E1 29740.629,E2 29740.629} C_VEL
LIN {X 0,Y 137.33,Z 942.978,A -85,B 0,C 180,E1 29761.959,E2 29761.959} C_VEL
LIN {X 0,Y 132.845,Z 949.637,A -85,B 0,C 180,E1 29776.832,E2 29776.832} C_VEL
LIN {X 0,Y 133.878,Z 951.766,A -85,B 0,C 180,E1 29790.018,E2 29790.018} C_VEL
LIN {X 0,Y 132.753,Z 949.633,A -85,B 0,C 180,E1 29803.214,E2 29803.214} C_VEL
LIN {X 0,Y 136.971,Z 942.075,A -85,B 0,C 180,E1 29819.51,E2 29819.51} C_VEL
LIN {X 0,Y 150.671,Z 928.375,A -85,B 0,C 180,E1 29834.767,E2 29834.767} C_VEL
LIN {X 0,Y 170.868,Z 909.499,A -85,B 0,C 180,E1 29846.262,E2 29846.262} C_VEL
LIN {X 0,Y 194.372,Z 885.271,A -85,B 0,C 180,E1 29854.604,E2 29854.604} C_VEL
LIN {X 0,Y 218.468,Z 855.785,A -85,B 0,C 180,E1 29860.487,E2 29860.487} C_VEL
LIN {X 0,Y 239.897,Z 823.072,A -85,B 0,C 180,E1 29864.378,E2 29864.378} C_VEL
LIN {X 0,Y 252.254,Z 799.072,A -85,B 0,C 180,E1 29866.336,E2 29866.336} C_VEL
LIN {X 0,Y 257.442,Z 778.411,A -85,B 0,C 180,E1 29870.62,E2 29870.62} C_VEL
LIN {X 0,Y 256.004,Z 770.89,A -85,B 0,C 180,E1 29876.603,E2 29876.603} C_VEL
LIN {X 0,Y 255.841,Z 768.069,A -85,B 0,C 180,E1 29879.996,E2 29879.996} C_VEL
LIN {X 0,Y 254.845,Z 769.454,A -85,B 0,C 180,E1 29885.111,E2 29885.111} C_VEL
LIN {X 0,Y 254.032,Z 775.284,A -85,B 0,C 180,E1 29891.171,E2 29891.171} C_VEL
LIN {X 0,Y 252.897,Z 786.217,A -85,B 0,C 180,E1 29897.423,E2 29897.423} C_VEL
LIN {X 0,Y 251.209,Z 796.747,A -85,B 0,C 180,E1 29901.735,E2 29901.735} C_VEL
LIN {X 0,Y 231.247,Z 828.211,A -85,B 0,C 180,E1 29905.694,E2 29905.694} C_VEL
LIN {X 0,Y 209.517,Z 854.965,A -85,B 0,C 180,E1 29910.797,E2 29910.797} C_VEL
LIN {X 0,Y 186.61,Z 877.873,A -85,B 0,C 180,E1 29917.804,E2 29917.804} C_VEL
LIN {X 0,Y 164.762,Z 896.093,A -85,B 0,C 180,E1 29927.562,E2 29927.562} C_VEL
LIN {X 0,Y 148.435,Z 908.12,A -85,B 0,C 180,E1 29939.291,E2 29939.291} C_VEL
LIN {X 0,Y 139.202,Z 914.501,A -85,B 0,C 180,E1 29950.922,E2 29950.922} C_VEL
LIN {X 0,Y 134.585,Z 917.813,A -85,B 0,C 180,E1 29968.361,E2 29968.361} C_VEL
LIN {X 0,Y 136.419,Z 916.397,A -85,B 0,C 180,E1 29982.598,E2 29982.598} C_VEL
LIN {X 0,Y 136.254,Z 915.315,A -85,B 0,C 180,E1 29988.099,E2 29988.099} C_VEL
LIN {X 0,Y 136.24,Z 912.611,A -85,B 0,C 180,E1 29996.382,E2 29996.382} C_VEL
LIN {X 0,Y 136.874,Z 912.164,A -85,B 0,C 180,E1 29997.247,E2 29997.247} C_VEL
LIN {X 0,Y 154.219,Z 900.463,A -85,B 0,C 180,E1 30011.523,E2 30011.523} C_VEL
LIN {X 0,Y 169.621,Z 888.948,A -85,B 0,C 180,E1 30019.328,E2 30019.328} C_VEL
LIN {X 0,Y 170.283,Z 887.821,A -85,B 0,C 180,E1 30020.409,E2 30020.409} C_VEL
LIN {X 0,Y 135.584,Z 898.109,A -85,B 0,C 180,E1 30040.425,E2 30040.425} C_VEL
LIN {X 0,Y 127.308,Z 907.075,A -85,B 0,C 180,E1 30066.843,E2 30066.843} C_VEL
LIN {X 0,Y 137.4,Z 924.372,A -85,B 0,C 180,E1 30082.707,E2 30082.707} C_VEL
LIN {X 0,Y 157.329,Z 936.721,A -85,B 0,C 180,E1 30096.237,E2 30096.237} C_VEL
LIN {X 0,Y 154.55,Z 937.485,A -85,B 0,C 180,E1 30098.367,E2 30098.367} C_VEL
LIN {X 0,Y 131.856,Z 940.43,A -85,B 0,C 180,E1 30117.864,E2 30117.864} C_VEL
LIN {X 0,Y 125.034,Z 948.617,A -85,B 0,C 180,E1 30135.993,E2 30135.993} C_VEL
LIN {X 0,Y 126.004,Z 950.774,A -85,B 0,C 180,E1 30150.019,E2 30150.019} C_VEL
LIN {X 0,Y 124.909,Z 948.61,A -85,B 0,C 180,E1 30164.06,E2 30164.06} C_VEL
LIN {X 0,Y 130.076,Z 940.802,A -85,B 0,C 180,E1 30181.635,E2 30181.635} C_VEL
LIN {X 0,Y 144.875,Z 927.279,A -85,B 0,C 180,E1 30197.088,E2 30197.088} C_VEL
LIN {X 0,Y 166.41,Z 908.356,A -85,B 0,C 180,E1 30208.635,E2 30208.635} C_VEL
LIN {X 0,Y 190.279,Z 884.864,A -85,B 0,C 180,E1 30216.663,E2 30216.663} C_VEL
LIN {X 0,Y 214.721,Z 856.068,A -85,B 0,C 180,E1 30222.333,E2 30222.333} C_VEL
LIN {X 0,Y 236.754,Z 823.586,A -85,B 0,C 180,E1 30226.118,E2 30226.118} C_VEL
LIN {X 0,Y 248.926,Z 800.752,A -85,B 0,C 180,E1 30228.068,E2 30228.068} C_VEL
LIN {X 0,Y 253.578,Z 784.864,A -85,B 0,C 180,E1 30231.406,E2 30231.406} C_VEL
LIN {X 0,Y 252.729,Z 778.273,A -85,B 0,C 180,E1 30236.559,E2 30236.559} C_VEL
LIN {X 0,Y 252.572,Z 775.368,A -85,B 0,C 180,E1 30239.996,E2 30239.996} C_VEL
LIN {X 0,Y 251.464,Z 776.747,A -85,B 0,C 180,E1 30245.18,E2 30245.18} C_VEL
LIN {X 0,Y 250.192,Z 782.825,A -85,B 0,C 180,E1 30251.345,E2 30251.345} C_VEL
LIN {X 0,Y 248.594,Z 792.693,A -85,B 0,C 180,E1 30256.971,E2 30256.971} C_VEL
LIN {X 0,Y 246.444,Z 801.385,A -85,B 0,C 180,E1 30260.507,E2 30260.507} C_VEL
LIN {X 0,Y 226.44,Z 831.412,A -85,B 0,C 180,E1 30264.232,E2 30264.232} C_VEL
LIN {X 0,Y 202.728,Z 859.106,A -85,B 0,C 180,E1 30269.65,E2 30269.65} C_VEL
LIN {X 0,Y 178.947,Z 881.404,A -85,B 0,C 180,E1 30276.905,E2 30276.905} C_VEL
LIN {X 0,Y 156.185,Z 899.174,A -85,B 0,C 180,E1 30287.206,E2 30287.206} C_VEL
LIN {X 0,Y 139.354,Z 910.669,A -85,B 0,C 180,E1 30300.002,E2 30300.002} C_VEL
LIN {X 0,Y 128.8,Z 917.394,A -85,B 0,C 180,E1 30316.373,E2 30316.373} C_VEL
LIN {X 0,Y 126.859,Z 918.896,A -85,B 0,C 180,E1 30329.981,E2 30329.981} C_VEL
LIN {X 0,Y 128.848,Z 917.352,A -85,B 0,C 180,E1 30343.584,E2 30343.584} C_VEL
LIN {X 0,Y 136.874,Z 912.164,A -85,B 0,C 180,E1 30357.247,E2 30357.247} C_VEL
LIN {X 0,Y 139.758,Z 908.699,A -85,B 0,C 180,E1 30364.274,E2 30364.274} C_VEL
LIN {X 0,Y 144.16,Z 904.311,A -85,B 0,C 180,E1 30370.928,E2 30370.928} C_VEL
LIN {X 0,Y 159.725,Z 893.571,A -85,B 0,C 180,E1 30379.345,E2 30379.345} C_VEL
LIN {X 0,Y 160.507,Z 892.599,A -85,B 0,C 180,E1 30380.353,E2 30380.353} C_VEL
LIN {X 0,Y 125.119,Z 903.256,A -85,B 0,C 180,E1 30404.533,E2 30404.533} C_VEL
LIN {X 0,Y 122.124,Z 912.827,A -85,B 0,C 180,E1 30433.458,E2 30433.458} C_VEL
LIN {X 0,Y 137.062,Z 929.291,A -85,B 0,C 180,E1 30449.835,E2 30449.835} C_VEL
LIN {X 0,Y 147.101,Z 935.001,A -85,B 0,C 180,E1 30456.023,E2 30456.023} C_VEL
LIN {X 0,Y 146.142,Z 935.823,A -85,B 0,C 180,E1 30457.857,E2 30457.857} C_VEL
LIN {X 0,Y 127.071,Z 937.725,A -85,B 0,C 180,E1 30473.425,E2 30473.425} C_VEL
LIN {X 0,Y 117.803,Z 946.47,A -85,B 0,C 180,E1 30491.264,E2 30491.264} C_VEL
LIN {X 0,Y 117.115,Z 949.099,A -85,B 0,C 180,E1 30502.587,E2 30502.587} C_VEL
LIN {X 0,Y 118.12,Z 949.78,A -85,B 0,C 180,E1 30510.02,E2 30510.02} C_VEL
LIN {X 0,Y 117.085,Z 947.584,A -85,B 0,C 180,E1 30525.021,E2 30525.021} C_VEL
LIN {X 0,Y 123.143,Z 939.742,A -85,B 0,C 180,E1 30543.644,E2 30543.644} C_VEL
LIN {X 0,Y 139.343,Z 926.171,A -85,B 0,C 180,E1 30559.594,E2 30559.594} C_VEL
LIN {X 0,Y 162.774,Z 906.713,A -85,B 0,C 180,E1 30571.379,E2 30571.379} C_VEL
LIN {X 0,Y 187.887,Z 882.893,A -85,B 0,C 180,E1 30579.203,E2 30579.203} C_VEL
LIN {X 0,Y 213.196,Z 853.829,A -85,B 0,C 180,E1 30584.6,E2 30584.6} C_VEL
LIN {X 0,Y 235.907,Z 820.758,A -85,B 0,C 180,E1 30588.203,E2 30588.203} C_VEL
LIN {X 0,Y 245.279,Z 803.759,A -85,B 0,C 180,E1 30589.566,E2 30589.566} C_VEL
LIN {X 0,Y 249.655,Z 790.843,A -85,B 0,C 180,E1 30592.347,E2 30592.347} C_VEL
LIN {X 0,Y 249.14,Z 783.977,A -85,B 0,C 180,E1 30598.253,E2 30598.253} C_VEL
LIN {X 0,Y 249.155,Z 782.586,A -85,B 0,C 180,E1 30599.996,E2 30599.996} C_VEL
LIN {X 0,Y 247.96,Z 783.624,A -85,B 0,C 180,E1 30604.811,E2 30604.811} C_VEL
LIN {X 0,Y 246.108,Z 790.315,A -85,B 0,C 180,E1 30611.536,E2 30611.536} C_VEL
LIN {X 0,Y 243.448,Z 801.529,A -85,B 0,C 180,E1 30617.654,E2 30617.654} C_VEL
LIN {X 0,Y 242.44,Z 804.748,A -85,B 0,C 180,E1 30619.012,E2 30619.012} C_VEL
LIN {X 0,Y 221.653,Z 834.621,A -85,B 0,C 180,E1 30622.731,E2 30622.731} C_VEL
LIN {X 0,Y 197.49,Z 861.709,A -85,B 0,C 180,E1 30628.051,E2 30628.051} C_VEL
LIN {X 0,Y 173.564,Z 883.095,A -85,B 0,C 180,E1 30635.103,E2 30635.103} C_VEL
LIN {X 0,Y 150.506,Z 900.211,A -85,B 0,C 180,E1 30645.171,E2 30645.171} C_VEL
LIN {X 0,Y 131.285,Z 912.515,A -85,B 0,C 180,E1 30659.664,E2 30659.664} C_VEL
LIN {X 0,Y 121.186,Z 918.386,A -85,B 0,C 180,E1 30675.498,E2 30675.498} C_VEL
LIN {X 0,Y 119.042,Z 919.881,A -85,B 0,C 180,E1 30689.98,E2 30689.98} C_VEL
LIN {X 0,Y 121.228,Z 918.347,A -85,B 0,C 180,E1 30704.456,E2 30704.456} C_VEL
LIN {X 0,Y 131.477,Z 912.305,A -85,B 0,C 180,E1 30720.469,E2 30720.469} C_VEL
LIN {X 0,Y 144.16,Z 904.311,A -85,B 0,C 180,E1 30730.928,E2 30730.928} C_VEL
LIN {X 0,Y 147.583,Z 901.014,A -85,B 0,C 180,E1 30735.139,E2 30735.139} C_VEL
LIN {X 0,Y 149.888,Z 897.826,A -85,B 0,C 180,E1 30739.536,E2 30739.536} C_VEL
LIN {X 0,Y 150.557,Z 897.155,A -85,B 0,C 180,E1 30740.328,E2 30740.328} C_VEL
LIN {X 0,Y 113.919,Z 909.227,A -85,B 0,C 180,E1 30772.368,E2 30772.368} C_VEL
LIN {X 0,Y 118.621,Z 918.144,A -85,B 0,C 180,E1 30800.57,E2 30800.57} C_VEL
LIN {X 0,Y 138.073,Z 933.444,A -85,B 0,C 180,E1 30816.449,E2 30816.449} C_VEL
LIN {X 0,Y 135.679,Z 934.034,A -85,B 0,C 180,E1 30818.609,E2 30818.609} C_VEL
LIN {X 0,Y 122.927,Z 935.02,A -85,B 0,C 180,E1 30828.8,E2 30828.8} C_VEL
LIN {X 0,Y 111.368,Z 944.121,A -85,B 0,C 180,E1 30845.934,E2 30845.934} C_VEL
LIN {X 0,Y 109.203,Z 948.092,A -85,B 0,C 180,E1 30862.047,E2 30862.047} C_VEL
LIN {X 0,Y 110.232,Z 948.785,A -85,B 0,C 180,E1 30870.022,E2 30870.022} C_VEL
LIN {X 0,Y 109.278,Z 946.556,A -85,B 0,C 180,E1 30886.123,E2 30886.123} C_VEL
LIN {X 0,Y 116.37,Z 938.683,A -85,B 0,C 180,E1 30905.894,E2 30905.894} C_VEL
LIN {X 0,Y 134.125,Z 925.069,A -85,B 0,C 180,E1 30922.288,E2 30922.288} C_VEL
LIN {X 0,Y 158.644,Z 905.853,A -85,B 0,C 180,E1 30933.899,E2 30933.899} C_VEL
LIN {X 0,Y 184.68,Z 882.162,A -85,B 0,C 180,E1 30941.496,E2 30941.496} C_VEL
LIN {X 0,Y 210.309,Z 853.638,A -85,B 0,C 180,E1 30946.613,E2 30946.613} C_VEL
LIN {X 0,Y 233.385,Z 821.113,A -85,B 0,C 180,E1 30950.028,E2 30950.028} C_VEL
LIN {X 0,Y 242.235,Z 805.54,A -85,B 0,C 180,E1 30951.377,E2 30951.377} C_VEL
LIN {X 0,Y 245.792,Z 795.627,A -85,B 0,C 180,E1 30953.804,E2 30953.804} C_VEL
LIN {X 0,Y 245.488,Z 789.69,A -85,B 0,C 180,E1 30959.996,E2 30959.996} C_VEL
LIN {X 0,Y 244.589,Z 789.895,A -85,B 0,C 180,E1 30963.546,E2 30963.546} C_VEL
LIN {X 0,Y 242.432,Z 795.233,A -85,B 0,C 180,E1 30969.891,E2 30969.891} C_VEL
LIN {X 0,Y 239.794,Z 804.261,A -85,B 0,C 180,E1 30975.521,E2 30975.521} C_VEL
LIN {X 0,Y 238.356,Z 808.509,A -85,B 0,C 180,E1 30977.501,E2 30977.501} C_VEL
LIN {X 0,Y 217.287,Z 837.47,A -85,B 0,C 180,E1 30981.113,E2 30981.113} C_VEL
LIN {X 0,Y 193.474,Z 863.228,A -85,B 0,C 180,E1 30986.116,E2 30986.116} C_VEL
LIN {X 0,Y 167.046,Z 885.826,A -85,B 0,C 180,E1 30993.648,E2 30993.648} C_VEL
LIN {X 0,Y 142.748,Z 902.668,A -85,B 0,C 180,E1 31004.211,E2 31004.211} C_VEL
LIN {X 0,Y 125.041,Z 913.234,A -85,B 0,C 180,E1 31017.346,E2 31017.346} C_VEL
LIN {X 0,Y 113.596,Z 919.38,A -85,B 0,C 180,E1 31034.506,E2 31034.506} C_VEL
LIN {X 0,Y 111.215,Z 920.868,A -85,B 0,C 180,E1 31049.978,E2 31049.978} C_VEL
LIN {X 0,Y 113.637,Z 919.343,A -85,B 0,C 180,E1 31065.445,E2 31065.445} C_VEL
LIN {X 0,Y 125.044,Z 913.137,A -85,B 0,C 180,E1 31082.608,E2 31082.608} C_VEL
LIN {X 0,Y 145.072,Z 901.1,A -85,B 0,C 180,E1 31096.956,E2 31096.956} C_VEL
LIN {X 0,Y 149.888,Z 897.826,A -85,B 0,C 180,E1 31099.536,E2 31099.536} C_VEL
LIN {X 0,Y 148.621,Z 897.432,A -85,B 0,C 180,E1 31101.522,E2 31101.522} C_VEL
LIN {X 0,Y 140.904,Z 899.707,A -85,B 0,C 180,E1 31104.134,E2 31104.134} C_VEL
LIN {X 0,Y 125.889,Z 904.991,A -85,B 0,C 180,E1 31108.29,E2 31108.29} C_VEL
LIN {X 0,Y 124.304,Z 905.454,A -85,B 0,C 180,E1 31109.225,E2 31109.225} C_VEL
LIN {X 0,Y 116.882,Z 922.932,A -85,B 0,C 180,E1 31168.034,E2 31168.034} C_VEL
LIN {X 0,Y 127.978,Z 930.878,A -85,B 0,C 180,E1 31176.299,E2 31176.299} C_VEL
LIN {X 0,Y 127.309,Z 931.651,A -85,B 0,C 180,E1 31178.18,E2 31178.18} C_VEL
LIN {X 0,Y 118.503,Z 932.924,A -85,B 0,C 180,E1 31184.826,E2 31184.826} C_VEL
LIN {X 0,Y 104.022,Z 943.085,A -85,B 0,C 180,E1 31204.114,E2 31204.114} C_VEL
LIN {X 0,Y 101.304,Z 947.082,A -85,B 0,C 180,E1 31221.422,E2 31221.422} C_VEL
LIN {X 0,Y 102.331,Z 947.789,A -85,B 0,C 180,E1 31230.023,E2 31230.023} C_VEL
LIN {X 0,Y 101.517,Z 945.529,A -85,B 0,C 180,E1 31247.393,E2 31247.393} C_VEL
LIN {X 0,Y 109.784,Z 937.612,A -85,B 0,C 180,E1 31268.423,E2 31268.423} C_VEL
LIN {X 0,Y 129.233,Z 923.982,A -85,B 0,C 180,E1 31285.189,E2 31285.189} C_VEL
LIN {X 0,Y 155.457,Z 904.485,A -85,B 0,C 180,E1 31296.745,E2 31296.745} C_VEL
LIN {X 0,Y 183.129,Z 880.103,A -85,B 0,C 180,E1 31304.171,E2 31304.171} C_VEL
LIN {X 0,Y 210.301,Z 850.375,A -85,B 0,C 180,E1 31309.073,E2 31309.073} C_VEL
LIN {X 0,Y 233.493,Z 817.704,A -85,B 0,C 180,E1 31312.201,E2 31312.201} C_VEL
LIN {X 0,Y 238.471,Z 809.337,A -85,B 0,C 180,E1 31312.798,E2 31312.798} C_VEL
LIN {X 0,Y 241.639,Z 801.665,A -85,B 0,C 180,E1 31314.6,E2 31314.6} C_VEL
LIN {X 0,Y 241.557,Z 796.643,A -85,B 0,C 180,E1 31319.995,E2 31319.995} C_VEL
LIN {X 0,Y 240.634,Z 796.944,A -85,B 0,C 180,E1 31323.605,E2 31323.605} C_VEL
LIN {X 0,Y 237.995,Z 802.469,A -85,B 0,C 180,E1 31330.076,E2 31330.076} C_VEL
LIN {X 0,Y 234.466,Z 812.154,A -85,B 0,C 180,E1 31335.877,E2 31335.877} C_VEL
LIN {X 0,Y 211.082,Z 842.701,A -85,B 0,C 180,E1 31339.773,E2 31339.773} C_VEL
LIN {X 0,Y 185.854,Z 868.16,A -85,B 0,C 180,E1 31344.987,E2 31344.987} C_VEL
LIN {X 0,Y 160.854,Z 888.334,A -85,B 0,C 180,E1 31352.001,E2 31352.001} C_VEL
LIN {X 0,Y 135.032,Z 905.126,A -85,B 0,C 180,E1 31363.141,E2 31363.141} C_VEL
LIN {X 0,Y 115.511,Z 915.717,A -85,B 0,C 180,E1 31378.328,E2 31378.328} C_VEL
LIN {X 0,Y 106.067,Z 920.373,A -85,B 0,C 180,E1 31393.375,E2 31393.375} C_VEL
LIN {X 0,Y 103.381,Z 921.856,A -85,B 0,C 180,E1 31409.977,E2 31409.977} C_VEL
LIN {X 0,Y 106.102,Z 920.337,A -85,B 0,C 180,E1 31426.572,E2 31426.572} C_VEL
LIN {X 0,Y 118.832,Z 913.958,A -85,B 0,C 180,E1 31444.99,E2 31444.99} C_VEL
LIN {X 0,Y 140.953,Z 901.462,A -85,B 0,C 180,E1 31459.856,E2 31459.856} C_VEL
LIN {X 0,Y 124.304,Z 905.454,A -85,B 0,C 180,E1 31469.225,E2 31469.225} C_VEL
LIN {X 0,Y 112.902,Z 909.306,A -85,B 0,C 180,E1 31475.401,E2 31475.401} C_VEL
LIN {X 0,Y 103.267,Z 912.998,A -85,B 0,C 180,E1 31482.896,E2 31482.896} C_VEL
LIN {X 0,Y 118.538,Z 928.228,A -85,B 0,C 180,E1 31536.46,E2 31536.46} C_VEL
LIN {X 0,Y 119.678,Z 928.942,A -85,B 0,C 180,E1 31537.19,E2 31537.19} C_VEL
LIN {X 0,Y 114.192,Z 931.103,A -85,B 0,C 180,E1 31540.97,E2 31540.97} C_VEL
LIN {X 0,Y 96.807,Z 942.057,A -85,B 0,C 180,E1 31562.023,E2 31562.023} C_VEL
LIN {X 0,Y 93.406,Z 946.072,A -85,B 0,C 180,E1 31580.69,E2 31580.69} C_VEL
LIN {X 0,Y 94.428,Z 946.793,A -85,B 0,C 180,E1 31590.025,E2 31590.025} C_VEL
LIN {X 0,Y 93.799,Z 944.499,A -85,B 0,C 180,E1 31608.876,E2 31608.876} C_VEL
LIN {X 0,Y 103.19,Z 936.71,A -85,B 0,C 180,E1 31630.953,E2 31630.953} C_VEL
LIN {X 0,Y 124.667,Z 922.887,A -85,B 0,C 180,E1 31648.333,E2 31648.333} C_VEL
LIN {X 0,Y 151.847,Z 903.76,A -85,B 0,C 180,E1 31659.468,E2 31659.468} C_VEL
LIN {X 0,Y 181.049,Z 878.94,A -85,B 0,C 180,E1 31666.687,E2 31666.687} C_VEL
LIN {X 0,Y 207.873,Z 850.369,A -85,B 0,C 180,E1 31671.148,E2 31671.148} C_VEL
LIN {X 0,Y 231.667,Z 817.814,A -85,B 0,C 180,E1 31674.097,E2 31674.097} C_VEL
LIN {X 0,Y 236.017,Z 810.48,A -85,B 0,C 180,E1 31674.798,E2 31674.798} C_VEL
LIN {X 0,Y 237.343,Z 807.325,A -85,B 0,C 180,E1 31675.748,E2 31675.748} C_VEL
LIN {X 0,Y 237.431,Z 803.509,A -85,B 0,C 180,E1 31679.995,E2 31679.995} C_VEL
LIN {X 0,Y 236.412,Z 803.844,A -85,B 0,C 180,E1 31683.669,E2 31683.669} C_VEL
LIN {X 0,Y 233.394,Z 809.451,A -85,B 0,C 180,E1 31690.114,E2 31690.114} C_VEL
LIN {X 0,Y 230.919,Z 815.09,A -85,B 0,C 180,E1 31693.729,E2 31693.729} C_VEL
LIN {X 0,Y 229.053,Z 818.05,A -85,B 0,C 180,E1 31694.554,E2 31694.554} C_VEL
LIN {X 0,Y 205.477,Z 847.135,A -85,B 0,C 180,E1 31698.266,E2 31698.266} C_VEL
LIN {X 0,Y 179.645,Z 871.908,A -85,B 0,C 180,E1 31703.44,E2 31703.44} C_VEL
LIN {X 0,Y 153.921,Z 891.32,A -85,B 0,C 180,E1 31710.501,E2 31710.501} C_VEL
LIN {X 0,Y 129.311,Z 906.426,A -85,B 0,C 180,E1 31720.866,E2 31720.866} C_VEL
LIN {X 0,Y 108.887,Z 916.728,A -85,B 0,C 180,E1 31736.151,E2 31736.151} C_VEL
LIN {X 0,Y 98.562,Z 921.369,A -85,B 0,C 180,E1 31752.068,E2 31752.068} C_VEL
LIN {X 0,Y 95.554,Z 922.842,A -85,B 0,C 180,E1 31769.975,E2 31769.975} C_VEL
LIN {X 0,Y 98.597,Z 921.332,A -85,B 0,C 180,E1 31787.874,E2 31787.874} C_VEL
LIN {X 0,Y 112.487,Z 914.966,A -85,B 0,C 180,E1 31807.285,E2 31807.285} C_VEL
LIN {X 0,Y 128.018,Z 906.995,A -85,B 0,C 180,E1 31818.348,E2 31818.348} C_VEL
LIN {X 0,Y 130.445,Z 905.403,A -85,B 0,C 180,E1 31820.351,E2 31820.351} C_VEL
LIN {X 0,Y 103.267,Z 912.998,A -85,B 0,C 180,E1 31842.896,E2 31842.896} C_VEL
LIN {X 0,Y 95.552,Z 916.741,A -85,B 0,C 180,E1 31851.738,E2 31851.738} C_VEL
LIN {X 0,Y 90.219,Z 920.421,A -85,B 0,C 180,E1 31861.835,E2 31861.835} C_VEL
LIN {X 0,Y 109.597,Z 929.363,A -85,B 0,C 180,E1 31896.731,E2 31896.731} C_VEL
LIN {X 0,Y 91.709,Z 939.782,A -85,B 0,C 180,E1 31915.703,E2 31915.703} C_VEL
LIN {X 0,Y 85.52,Z 945.063,A -85,B 0,C 180,E1 31939.823,E2 31939.823} C_VEL
LIN {X 0,Y 86.492,Z 945.792,A -85,B 0,C 180,E1 31950.028,E2 31950.028} C_VEL
LIN {X 0,Y 86.156,Z 943.469,A -85,B 0,C 180,E1 31970.623,E2 31970.623} C_VEL
LIN {X 0,Y 96.91,Z 935.786,A -85,B 0,C 180,E1 31993.881,E2 31993.881} C_VEL
LIN {X 0,Y 120.52,Z 921.779,A -85,B 0,C 180,E1 32011.691,E2 32011.691} C_VEL
LIN {X 0,Y 149.303,Z 902.481,A -85,B 0,C 180,E1 32022.539,E2 32022.539} C_VEL
LIN {X 0,Y 179.326,Z 877.77,A -85,B 0,C 180,E1 32029.259,E2 32029.259} C_VEL
LIN {X 0,Y 207.575,Z 848.221,A -85,B 0,C 180,E1 32033.514,E2 32033.514} C_VEL
